LIN {X 0,Y 411.249,Z 344.255,A -85,B 0,C 180,E1 -10637.915,E2 -10637.915} C_VEL
LIN {X 0,Y 411.2,Z 344.267,A -85,B 0,C 180,E1 -10641.034,E2 -10641.034} C_VEL
LIN {X 0,Y 411.23,Z 344.259,A -85,B 0,C 180,E1 -10644.215,E2 -10644.215} C_VEL
LIN {X 0,Y 411.262,Z 344.258,A -85,B 0,C 180,E1 -10647.477,E2 -10647.477} C_VEL
LIN {X 0,Y 411.192,Z 344.266,A -85,B 0,C 180,E1 -10650.847,E2 -10650.847} C_VEL
LIN {X 0,Y 411.208,Z 344.262,A -85,B 0,C 180,E1 -10654.333,E2 -10654.333} C_VEL
LIN {X 0,Y 411.206,Z 344.261,A -85,B 0,C 180,E1 -10657.972,E2 -10657.972} C_VEL
LIN {X 0,Y 411.202,Z 344.264,A -85,B 0,C 180,E1 -10661.234,E2 -10661.234} C_VEL
LIN {X 0,Y 411.179,Z 344.268,A -85,B 0,C 180,E1 -10664.49,E2 -10664.49} C_VEL
LIN {X 0,Y 411.181,Z 344.267,A -85,B 0,C 180,E1 -10668.195,E2 -10668.195} C_VEL
LIN {X 0,Y 411.221,Z 344.265,A -85,B 0,C 180,E1 -10670.776,E2 -10670.776} C_VEL
LIN {X 0,Y 411.199,Z 344.267,A -85,B 0,C 180,E1 -10674.471,E2 -10674.471} C_VEL
LIN {X 0,Y 411.208,Z 344.263,A -85,B 0,C 180,E1 -10676.873,E2 -10676.873} C_VEL
LIN {X 0,Y 411.234,Z 344.26,A -85,B 0,C 180,E1 -10680.644,E2 -10680.644} C_VEL
LIN {X 0,Y 411.239,Z 344.259,A -85,B 0,C 180,E1 -10683.619,E2 -10683.619} C_VEL
LIN {X 0,Y 411.204,Z 344.264,A -85,B 0,C 180,E1 -10686.852,E2 -10686.852} C_VEL
LIN {X 0,Y 411.265,Z 344.256,A -85,B 0,C 180,E1 -10690.031,E2 -10690.031} C_VEL
LIN {X 0,Y 411.264,Z 344.254,A -85,B 0,C 180,E1 -10693.131,E2 -10693.131} C_VEL
LIN {X 0,Y 411.306,Z 344.251,A -85,B 0,C 180,E1 -10696.896,E2 -10696.896} C_VEL
LIN {X 0,Y 411.294,Z 344.253,A -85,B 0,C 180,E1 -10700.161,E2 -10700.161} C_VEL
LIN {X 0,Y 411.453,Z 344.232,A -85,B 0,C 180,E1 -10703.133,E2 -10703.133} C_VEL
LIN {X 0,Y 411.311,Z 344.249,A -85,B 0,C 180,E1 -10705.099,E2 -10705.099} C_VEL
LIN {X 0,Y 411.515,Z 344.228,A -85,B 0,C 180,E1 -10708.043,E2 -10708.043} C_VEL
LIN {X 0,Y 411.641,Z 344.212,A -85,B 0,C 180,E1 -10710,E2 -10710} C_VEL
LIN {X 0,Y 411.468,Z 344.229,A -85,B 0,C 180,E1 -10712.937,E2 -10712.937} C_VEL
LIN {X 0,Y 411.453,Z 344.232,A -85,B 0,C 180,E1 -10716.867,E2 -10716.867} C_VEL
LIN {X 0,Y 411.295,Z 344.253,A -85,B 0,C 180,E1 -10719.839,E2 -10719.839} C_VEL
LIN {X 0,Y 411.306,Z 344.25,A -85,B 0,C 180,E1 -10723.104,E2 -10723.104} C_VEL
LIN {X 0,Y 411.25,Z 344.255,A -85,B 0,C 180,E1 -10725.055,E2 -10725.055} C_VEL
LIN {X 0,Y 410.564,Z 344.346,A -85,B 0,C 180,E1 -10725.872,E2 -10725.872} C_VEL
LIN {X 0,Y 407.698,Z 344.703,A -85,B 0,C 180,E1 -10727.2,E2 -10727.2} C_VEL
LIN {X 0,Y 405.284,Z 345.005,A -85,B 0,C 180,E1 -10728.272,E2 -10728.272} C_VEL
LIN {X 0,Y 404.249,Z 345.131,A -85,B 0,C 180,E1 -10729.101,E2 -10729.101} C_VEL
LIN {X 0,Y 404.166,Z 345.14,A -85,B 0,C 180,E1 -10729.382,E2 -10729.382} C_VEL
LIN {X 0,Y 404.157,Z 345.141,A -85,B 0,C 180,E1 -10732.834,E2 -10732.834} C_VEL
LIN {X 0,Y 404.185,Z 345.139,A -85,B 0,C 180,E1 -10735.767,E2 -10735.767} C_VEL
LIN {X 0,Y 404.197,Z 345.137,A -85,B 0,C 180,E1 -10738,E2 -10738} C_VEL
LIN {X 0,Y 404.141,Z 345.146,A -85,B 0,C 180,E1 -10741.558,E2 -10741.558} C_VEL
LIN {X 0,Y 404.186,Z 345.137,A -85,B 0,C 180,E1 -10745.016,E2 -10745.016} C_VEL
LIN {X 0,Y 404.158,Z 345.141,A -85,B 0,C 180,E1 -10748.757,E2 -10748.757} C_VEL
LIN {X 0,Y 404.191,Z 345.138,A -85,B 0,C 180,E1 -10751.611,E2 -10751.611} C_VEL
LIN {X 0,Y 404.195,Z 345.136,A -85,B 0,C 180,E1 -10754.529,E2 -10754.529} C_VEL
LIN {X 0,Y 404.139,Z 345.146,A -85,B 0,C 180,E1 -10757.296,E2 -10757.296} C_VEL
LIN {X 0,Y 404.171,Z 345.137,A -85,B 0,C 180,E1 -10759.956,E2 -10759.956} C_VEL
LIN {X 0,Y 404.139,Z 345.146,A -85,B 0,C 180,E1 -10763.125,E2 -10763.125} C_VEL
LIN {X 0,Y 404.148,Z 345.141,A -85,B 0,C 180,E1 -10766.188,E2 -10766.188} C_VEL
LIN {X 0,Y 404.149,Z 345.142,A -85,B 0,C 180,E1 -10769.715,E2 -10769.715} C_VEL
LIN {X 0,Y 404.199,Z 345.138,A -85,B 0,C 180,E1 -10773.123,E2 -10773.123} C_VEL
LIN {X 0,Y 404.181,Z 345.139,A -85,B 0,C 180,E1 -10775.335,E2 -10775.335} C_VEL
LIN {X 0,Y 404.143,Z 345.143,A -85,B 0,C 180,E1 -10778.581,E2 -10778.581} C_VEL
LIN {X 0,Y 404.214,Z 345.132,A -85,B 0,C 180,E1 -10781.762,E2 -10781.762} C_VEL
LIN {X 0,Y 404.211,Z 345.135,A -85,B 0,C 180,E1 -10784.882,E2 -10784.882} C_VEL
LIN {X 0,Y 404.262,Z 345.128,A -85,B 0,C 180,E1 -10787.959,E2 -10787.959} C_VEL
LIN {X 0,Y 404.438,Z 345.106,A -85,B 0,C 180,E1 -10792.1,E2 -10792.1} C_VEL
LIN {X 0,Y 404.429,Z 345.107,A -85,B 0,C 180,E1 -10794.015,E2 -10794.015} C_VEL
LIN {X 0,Y 404.485,Z 345.099,A -85,B 0,C 180,E1 -10798.009,E2 -10798.009} C_VEL
LIN {X 0,Y 404.615,Z 345.084,A -85,B 0,C 180,E1 -10800,E2 -10800} C_VEL
LIN {X 0,Y 404.427,Z 345.108,A -85,B 0,C 180,E1 -10802.989,E2 -10802.989} C_VEL
LIN {X 0,Y 404.419,Z 345.11,A -85,B 0,C 180,E1 -10805.985,E2 -10805.985} C_VEL
LIN {X 0,Y 404.271,Z 345.127,A -85,B 0,C 180,E1 -10809.002,E2 -10809.002} C_VEL
LIN {X 0,Y 404.261,Z 345.129,A -85,B 0,C 180,E1 -10812.042,E2 -10812.042} C_VEL
LIN {X 0,Y 404.212,Z 345.132,A -85,B 0,C 180,E1 -10815.118,E2 -10815.118} C_VEL
LIN {X 0,Y 404.216,Z 345.136,A -85,B 0,C 180,E1 -10818.238,E2 -10818.238} C_VEL
LIN {X 0,Y 404.144,Z 345.143,A -85,B 0,C 180,E1 -10821.419,E2 -10821.419} C_VEL
LIN {X 0,Y 404.182,Z 345.139,A -85,B 0,C 180,E1 -10824.666,E2 -10824.666} C_VEL
LIN {X 0,Y 404.2,Z 345.137,A -85,B 0,C 180,E1 -10828,E2 -10828} C_VEL
LIN {X 0,Y 404.144,Z 345.142,A -85,B 0,C 180,E1 -10831.558,E2 -10831.558} C_VEL
LIN {X 0,Y 404.19,Z 345.135,A -85,B 0,C 180,E1 -10835.016,E2 -10835.016} C_VEL
LIN {X 0,Y 404.162,Z 345.14,A -85,B 0,C 180,E1 -10838.756,E2 -10838.756} C_VEL
LIN {X 0,Y 404.127,Z 345.146,A -85,B 0,C 180,E1 -10841.6,E2 -10841.6} C_VEL
LIN {X 0,Y 404.15,Z 345.145,A -85,B 0,C 180,E1 -10844.522,E2 -10844.522} C_VEL
LIN {X 0,Y 404.137,Z 345.204,A -85,B 0,C 180,E1 -10846.378,E2 -10846.378} C_VEL
LIN {X 0,Y 406.071,Z 354.648,A -85,B 0,C 180,E1 -10849.599,E2 -10849.599} C_VEL
LIN {X 0,Y 407.763,Z 363.407,A -85,B 0,C 180,E1 -10852.451,E2 -10852.451} C_VEL
LIN {X 0,Y 407.874,Z 366.908,A -85,B 0,C 180,E1 -10853.525,E2 -10853.525} C_VEL
LIN {X 0,Y 406.615,Z 380.772,A -85,B 0,C 180,E1 -10857.601,E2 -10857.601} C_VEL
LIN {X 0,Y 405.74,Z 392.561,A -85,B 0,C 180,E1 -10860.987,E2 -10860.987} C_VEL
LIN {X 0,Y 404.928,Z 405.007,A -85,B 0,C 180,E1 -10864.492,E2 -10864.492} C_VEL
LIN {X 0,Y 404.265,Z 417.836,A -85,B 0,C 180,E1 -10868.051,E2 -10868.051} C_VEL
LIN {X 0,Y 403.765,Z 431.296,A -85,B 0,C 180,E1 -10871.741,E2 -10871.741} C_VEL
LIN {X 0,Y 403.666,Z 434.163,A -85,B 0,C 180,E1 -10872.522,E2 -10872.522} C_VEL
LIN {X 0,Y 404.99,Z 448.876,A -85,B 0,C 180,E1 -10873.06,E2 -10873.06} C_VEL
LIN {X 0,Y 405.875,Z 461.695,A -85,B 0,C 180,E1 -10873.716,E2 -10873.716} C_VEL
LIN {X 0,Y 406.362,Z 472.774,A -85,B 0,C 180,E1 -10874.45,E2 -10874.45} C_VEL
LIN {X 0,Y 405.508,Z 484.977,A -85,B 0,C 180,E1 -10875.445,E2 -10875.445} C_VEL
LIN {X 0,Y 404.832,Z 495.687,A -85,B 0,C 180,E1 -10876.54,E2 -10876.54} C_VEL
LIN {X 0,Y 404.282,Z 504.941,A -85,B 0,C 180,E1 -10877.704,E2 -10877.704} C_VEL
LIN {X 0,Y 403.773,Z 514.717,A -85,B 0,C 180,E1 -10879.216,E2 -10879.216} C_VEL
LIN {X 0,Y 403.451,Z 522.561,A -85,B 0,C 180,E1 -10880.727,E2 -10880.727} C_VEL
LIN {X 0,Y 403.419,Z 527.916,A -85,B 0,C 180,E1 -10881.989,E2 -10881.989} C_VEL
LIN {X 0,Y 403.454,Z 533.164,A -85,B 0,C 180,E1 -10883.528,E2 -10883.528} C_VEL
LIN {X 0,Y 403.546,Z 537.03,A -85,B 0,C 180,E1 -10885.004,E2 -10885.004} C_VEL
LIN {X 0,Y 403.598,Z 539.018,A -85,B 0,C 180,E1 -10886.006,E2 -10886.006} C_VEL
LIN {X 0,Y 403.599,Z 540.55,A -85,B 0,C 180,E1 -10887.005,E2 -10887.005} C_VEL
LIN {X 0,Y 403.628,Z 541.647,A -85,B 0,C 180,E1 -10888.004,E2 -10888.004} C_VEL
LIN {X 0,Y 403.761,Z 542.278,A -85,B 0,C 180,E1 -10889.003,E2 -10889.003} C_VEL
LIN {X 0,Y 403.888,Z 542.48,A -85,B 0,C 180,E1 -10890,E2 -10890} C_VEL
LIN {X 0,Y 403.869,Z 542.237,A -85,B 0,C 180,E1 -10890.997,E2 -10890.997} C_VEL
LIN {X 0,Y 403.64,Z 541.526,A -85,B 0,C 180,E1 -10891.996,E2 -10891.996} C_VEL
LIN {X 0,Y 403.621,Z 540.374,A -85,B 0,C 180,E1 -10892.994,E2 -10892.994} C_VEL
LIN {X 0,Y 403.642,Z 537.838,A -85,B 0,C 180,E1 -10894.494,E2 -10894.494} C_VEL
LIN {X 0,Y 403.478,Z 534.22,A -85,B 0,C 180,E1 -10895.999,E2 -10895.999} C_VEL
LIN {X 0,Y 403.406,Z 529.478,A -85,B 0,C 180,E1 -10897.508,E2 -10897.508} C_VEL
LIN {X 0,Y 403.451,Z 523.498,A -85,B 0,C 180,E1 -10899.02,E2 -10899.02} C_VEL
LIN {X 0,Y 403.678,Z 516.15,A -85,B 0,C 180,E1 -10900.533,E2 -10900.533} C_VEL
LIN {X 0,Y 404.112,Z 507.171,A -85,B 0,C 180,E1 -10902.046,E2 -10902.046} C_VEL
LIN {X 0,Y 404.701,Z 497.278,A -85,B 0,C 180,E1 -10903.41,E2 -10903.41} C_VEL
LIN {X 0,Y 405.648,Z 486.03,A -85,B 0,C 180,E1 -10904.678,E2 -10904.678} C_VEL
LIN {X 0,Y 406.71,Z 473.812,A -85,B 0,C 180,E1 -10905.793,E2 -10905.793} C_VEL
LIN {X 0,Y 406.567,Z 460.164,A -85,B 0,C 180,E1 -10906.831,E2 -10906.831} C_VEL
LIN {X 0,Y 406.397,Z 447.657,A -85,B 0,C 180,E1 -10907.59,E2 -10907.59} C_VEL
LIN {X 0,Y 405.002,Z 433.311,A -85,B 0,C 180,E1 -10908.316,E2 -10908.316} C_VEL
LIN {X 0,Y 403.649,Z 424.626,A -85,B 0,C 180,E1 -10908.725,E2 -10908.725} C_VEL
LIN {X 0,Y 403.913,Z 413.212,A -85,B 0,C 180,E1 -10911.7,E2 -10911.7} C_VEL
LIN {X 0,Y 404.396,Z 399.615,A -85,B 0,C 180,E1 -10915.35,E2 -10915.35} C_VEL
LIN {X 0,Y 405,Z 386.397,A -85,B 0,C 180,E1 -10919.071,E2 -10919.071} C_VEL
LIN {X 0,Y 405.793,Z 375.051,A -85,B 0,C 180,E1 -10922.473,E2 -10922.473} C_VEL
LIN {X 0,Y 407.226,Z 362.64,A -85,B 0,C 180,E1 -10926.542,E2 -10926.542} C_VEL
LIN {X 0,Y 406.953,Z 359.119,A -85,B 0,C 180,E1 -10927.88,E2 -10927.88} C_VEL
LIN {X 0,Y 405.885,Z 353.328,A -85,B 0,C 180,E1 -10930.37,E2 -10930.37} C_VEL
LIN {X 0,Y 404.721,Z 347.779,A -85,B 0,C 180,E1 -10933.169,E2 -10933.169} C_VEL
LIN {X 0,Y 404.136,Z 345.147,A -85,B 0,C 180,E1 -10934.782,E2 -10934.782} C_VEL
LIN {X 0,Y 404.14,Z 345.146,A -85,B 0,C 180,E1 -10937.296,E2 -10937.296} C_VEL
LIN {X 0,Y 404.172,Z 345.142,A -85,B 0,C 180,E1 -10939.955,E2 -10939.955} C_VEL
LIN {X 0,Y 404.143,Z 345.145,A -85,B 0,C 180,E1 -10943.124,E2 -10943.124} C_VEL
LIN {X 0,Y 404.149,Z 345.144,A -85,B 0,C 180,E1 -10946.188,E2 -10946.188} C_VEL
LIN {X 0,Y 404.149,Z 345.144,A -85,B 0,C 180,E1 -10949.715,E2 -10949.715} C_VEL
LIN {X 0,Y 404.198,Z 345.136,A -85,B 0,C 180,E1 -10953.123,E2 -10953.123} C_VEL
LIN {X 0,Y 404.18,Z 345.139,A -85,B 0,C 180,E1 -10955.334,E2 -10955.334} C_VEL
LIN {X 0,Y 404.143,Z 345.145,A -85,B 0,C 180,E1 -10958.581,E2 -10958.581} C_VEL
LIN {X 0,Y 404.207,Z 345.241,A -85,B 0,C 180,E1 -10961.089,E2 -10961.089} C_VEL
LIN {X 0,Y 408.313,Z 356.062,A -85,B 0,C 180,E1 -10962.076,E2 -10962.076} C_VEL
LIN {X 0,Y 410.568,Z 363.518,A -85,B 0,C 180,E1 -10962.816,E2 -10962.816} C_VEL
LIN {X 0,Y 409.73,Z 376.006,A -85,B 0,C 180,E1 -10963.93,E2 -10963.93} C_VEL
LIN {X 0,Y 408.903,Z 386.087,A -85,B 0,C 180,E1 -10965.06,E2 -10965.06} C_VEL
LIN {X 0,Y 408.091,Z 395.094,A -85,B 0,C 180,E1 -10966.302,E2 -10966.302} C_VEL
LIN {X 0,Y 407.321,Z 402.523,A -85,B 0,C 180,E1 -10967.545,E2 -10967.545} C_VEL
LIN {X 0,Y 406.546,Z 409.803,A -85,B 0,C 180,E1 -10969.038,E2 -10969.038} C_VEL
LIN {X 0,Y 405.811,Z 416.513,A -85,B 0,C 180,E1 -10970.807,E2 -10970.807} C_VEL
LIN {X 0,Y 405.237,Z 421.446,A -85,B 0,C 180,E1 -10972.526,E2 -10972.526} C_VEL
LIN {X 0,Y 404.71,Z 424.575,A -85,B 0,C 180,E1 -10974.019,E2 -10974.019} C_VEL
LIN {X 0,Y 404.488,Z 426.074,A -85,B 0,C 180,E1 -10975.016,E2 -10975.016} C_VEL
LIN {X 0,Y 404.384,Z 427.144,A -85,B 0,C 180,E1 -10976.014,E2 -10976.014} C_VEL
LIN {X 0,Y 404.257,Z 427.831,A -85,B 0,C 180,E1 -10977.01,E2 -10977.01} C_VEL
LIN {X 0,Y 404.21,Z 428.103,A -85,B 0,C 180,E1 -10978.007,E2 -10978.007} C_VEL
LIN {X 0,Y 404.089,Z 427.417,A -85,B 0,C 180,E1 -10980,E2 -10980} C_VEL
LIN {X 0,Y 403.974,Z 426.508,A -85,B 0,C 180,E1 -10980.997,E2 -10980.997} C_VEL
LIN {X 0,Y 404.062,Z 425.133,A -85,B 0,C 180,E1 -10981.993,E2 -10981.993} C_VEL
LIN {X 0,Y 404.164,Z 422.298,A -85,B 0,C 180,E1 -10983.489,E2 -10983.489} C_VEL
LIN {X 0,Y 404.29,Z 418.443,A -85,B 0,C 180,E1 -10984.986,E2 -10984.986} C_VEL
LIN {X 0,Y 404.663,Z 413.44,A -85,B 0,C 180,E1 -10986.482,E2 -10986.482} C_VEL
LIN {X 0,Y 405.124,Z 407.168,A -85,B 0,C 180,E1 -10987.977,E2 -10987.977} C_VEL
LIN {X 0,Y 405.514,Z 399.438,A -85,B 0,C 180,E1 -10989.476,E2 -10989.476} C_VEL
LIN {X 0,Y 405.938,Z 391.594,A -85,B 0,C 180,E1 -10990.726,E2 -10990.726} C_VEL
LIN {X 0,Y 406.574,Z 382.084,A -85,B 0,C 180,E1 -10991.972,E2 -10991.972} C_VEL
LIN {X 0,Y 407.198,Z 370.353,A -85,B 0,C 180,E1 -10993.22,E2 -10993.22} C_VEL
LIN {X 0,Y 407.582,Z 360.495,A -85,B 0,C 180,E1 -10994.072,E2 -10994.072} C_VEL
LIN {X 0,Y 407.621,Z 358.036,A -85,B 0,C 180,E1 -10994.26,E2 -10994.26} C_VEL
LIN {X 0,Y 404.235,Z 345.134,A -85,B 0,C 180,E1 -10995.246,E2 -10995.246} C_VEL
LIN {X 0,Y 404.208,Z 345.132,A -85,B 0,C 180,E1 -10998.238,E2 -10998.238} C_VEL
LIN {X 0,Y 404.142,Z 345.143,A -85,B 0,C 180,E1 -11001.419,E2 -11001.419} C_VEL
LIN {X 0,Y 404.18,Z 345.14,A -85,B 0,C 180,E1 -11004.665,E2 -11004.665} C_VEL
LIN {X 0,Y 404.198,Z 345.135,A -85,B 0,C 180,E1 -11007.999,E2 -11007.999} C_VEL
LIN {X 0,Y 404.142,Z 345.143,A -85,B 0,C 180,E1 -11011.558,E2 -11011.558} C_VEL
LIN {X 0,Y 404.187,Z 345.14,A -85,B 0,C 180,E1 -11015.016,E2 -11015.016} C_VEL
LIN {X 0,Y 404.166,Z 345.143,A -85,B 0,C 180,E1 -11018.756,E2 -11018.756} C_VEL
LIN {X 0,Y 404.152,Z 345.141,A -85,B 0,C 180,E1 -11021.604,E2 -11021.604} C_VEL
LIN {X 0,Y 404.148,Z 345.144,A -85,B 0,C 180,E1 -11024.522,E2 -11024.522} C_VEL
LIN {X 0,Y 404.142,Z 345.143,A -85,B 0,C 180,E1 -11027.296,E2 -11027.296} C_VEL
LIN {X 0,Y 404.17,Z 345.139,A -85,B 0,C 180,E1 -11029.955,E2 -11029.955} C_VEL
LIN {X 0,Y 404.138,Z 345.142,A -85,B 0,C 180,E1 -11033.125,E2 -11033.125} C_VEL
LIN {X 0,Y 404.146,Z 345.143,A -85,B 0,C 180,E1 -11036.188,E2 -11036.188} C_VEL
LIN {X 0,Y 404.147,Z 345.142,A -85,B 0,C 180,E1 -11039.715,E2 -11039.715} C_VEL
LIN {X 0,Y 404.196,Z 345.136,A -85,B 0,C 180,E1 -11043.123,E2 -11043.123} C_VEL
LIN {X 0,Y 404.178,Z 345.138,A -85,B 0,C 180,E1 -11045.334,E2 -11045.334} C_VEL
LIN {X 0,Y 404.164,Z 345.143,A -85,B 0,C 180,E1 -11048.582,E2 -11048.582} C_VEL
LIN {X 0,Y 404.215,Z 345.132,A -85,B 0,C 180,E1 -11051.762,E2 -11051.762} C_VEL
LIN {X 0,Y 404.207,Z 345.134,A -85,B 0,C 180,E1 -11054.882,E2 -11054.882} C_VEL
LIN {X 0,Y 404.258,Z 345.131,A -85,B 0,C 180,E1 -11057.959,E2 -11057.959} C_VEL
LIN {X 0,Y 404.405,Z 345.111,A -85,B 0,C 180,E1 -11062.129,E2 -11062.129} C_VEL
LIN {X 0,Y 404.421,Z 345.109,A -85,B 0,C 180,E1 -11064.015,E2 -11064.015} C_VEL
LIN {X 0,Y 404.484,Z 345.103,A -85,B 0,C 180,E1 -11068.009,E2 -11068.009} C_VEL
LIN {X 0,Y 404.611,Z 345.088,A -85,B 0,C 180,E1 -11070,E2 -11070} C_VEL
LIN {X 0,Y 404.425,Z 345.106,A -85,B 0,C 180,E1 -11072.988,E2 -11072.988} C_VEL
LIN {X 0,Y 404.4,Z 345.11,A -85,B 0,C 180,E1 -11076.988,E2 -11076.988} C_VEL
LIN {X 0,Y 404.26,Z 345.13,A -85,B 0,C 180,E1 -11080.012,E2 -11080.012} C_VEL
LIN {X 0,Y 404.267,Z 345.127,A -85,B 0,C 180,E1 -11083.212,E2 -11083.212} C_VEL
LIN {X 0,Y 404.217,Z 345.131,A -85,B 0,C 180,E1 -11087.007,E2 -11087.007} C_VEL
LIN {X 0,Y 404.166,Z 345.14,A -85,B 0,C 180,E1 -11089.382,E2 -11089.382} C_VEL
LIN {X 0,Y 403.495,Z 345.223,A -85,B 0,C 180,E1 -11090.213,E2 -11090.213} C_VEL
LIN {X 0,Y 400.631,Z 345.583,A -85,B 0,C 180,E1 -11091.564,E2 -11091.564} C_VEL
LIN {X 0,Y 398.217,Z 345.881,A -85,B 0,C 180,E1 -11092.655,E2 -11092.655} C_VEL
LIN {X 0,Y 397.198,Z 346.01,A -85,B 0,C 180,E1 -11093.499,E2 -11093.499} C_VEL
LIN {X 0,Y 397.124,Z 346.017,A -85,B 0,C 180,E1 -11093.785,E2 -11093.785} C_VEL
LIN {X 0,Y 397.196,Z 346.009,A -85,B 0,C 180,E1 -11097.39,E2 -11097.39} C_VEL
LIN {X 0,Y 397.08,Z 346.022,A -85,B 0,C 180,E1 -11100.883,E2 -11100.883} C_VEL
LIN {X 0,Y 397.127,Z 346.014,A -85,B 0,C 180,E1 -11104.494,E2 -11104.494} C_VEL
LIN {X 0,Y 397.105,Z 346.018,A -85,B 0,C 180,E1 -11108.275,E2 -11108.275} C_VEL
LIN {X 0,Y 397.157,Z 346.013,A -85,B 0,C 180,E1 -11111.993,E2 -11111.993} C_VEL
LIN {X 0,Y 397.114,Z 346.02,A -85,B 0,C 180,E1 -11115.065,E2 -11115.065} C_VEL
LIN {X 0,Y 397.068,Z 346.023,A -85,B 0,C 180,E1 -11118.021,E2 -11118.021} C_VEL
LIN {X 0,Y 397.132,Z 346.019,A -85,B 0,C 180,E1 -11121.139,E2 -11121.139} C_VEL
LIN {X 0,Y 397.122,Z 346.017,A -85,B 0,C 180,E1 -11124.497,E2 -11124.497} C_VEL
LIN {X 0,Y 397.081,Z 346.022,A -85,B 0,C 180,E1 -11127.929,E2 -11127.929} C_VEL
LIN {X 0,Y 397.126,Z 346.018,A -85,B 0,C 180,E1 -11131.457,E2 -11131.457} C_VEL
LIN {X 0,Y 397.157,Z 346.014,A -85,B 0,C 180,E1 -11134.488,E2 -11134.488} C_VEL
LIN {X 0,Y 397.113,Z 346.021,A -85,B 0,C 180,E1 -11137.086,E2 -11137.086} C_VEL
LIN {X 0,Y 397.152,Z 346.013,A -85,B 0,C 180,E1 -11140.353,E2 -11140.353} C_VEL
LIN {X 0,Y 397.171,Z 346.01,A -85,B 0,C 180,E1 -11143.553,E2 -11143.553} C_VEL
LIN {X 0,Y 397.233,Z 346.005,A -85,B 0,C 180,E1 -11146.703,E2 -11146.703} C_VEL
LIN {X 0,Y 397.223,Z 346.004,A -85,B 0,C 180,E1 -11149.809,E2 -11149.809} C_VEL
LIN {X 0,Y 397.369,Z 345.989,A -85,B 0,C 180,E1 -11152.888,E2 -11152.888} C_VEL
LIN {X 0,Y 397.258,Z 346.001,A -85,B 0,C 180,E1 -11154.925,E2 -11154.925} C_VEL
LIN {X 0,Y 397.454,Z 345.975,A -85,B 0,C 180,E1 -11157.973,E2 -11157.973} C_VEL
LIN {X 0,Y 397.584,Z 345.96,A -85,B 0,C 180,E1 -11160,E2 -11160} C_VEL
LIN {X 0,Y 397.386,Z 345.985,A -85,B 0,C 180,E1 -11163.042,E2 -11163.042} C_VEL
LIN {X 0,Y 397.369,Z 345.988,A -85,B 0,C 180,E1 -11166.092,E2 -11166.092} C_VEL
LIN {X 0,Y 397.241,Z 346.002,A -85,B 0,C 180,E1 -11169.162,E2 -11169.162} C_VEL
LIN {X 0,Y 397.224,Z 346.007,A -85,B 0,C 180,E1 -11172.258,E2 -11172.258} C_VEL
LIN {X 0,Y 397.184,Z 346.007,A -85,B 0,C 180,E1 -11175.392,E2 -11175.392} C_VEL
LIN {X 0,Y 397.168,Z 346.012,A -85,B 0,C 180,E1 -11178.573,E2 -11178.573} C_VEL
LIN {X 0,Y 397.102,Z 346.022,A -85,B 0,C 180,E1 -11181.818,E2 -11181.818} C_VEL
LIN {X 0,Y 397.161,Z 346.012,A -85,B 0,C 180,E1 -11185.132,E2 -11185.132} C_VEL
LIN {X 0,Y 397.166,Z 346.013,A -85,B 0,C 180,E1 -11187.776,E2 -11187.776} C_VEL
LIN {X 0,Y 397.083,Z 346.02,A -85,B 0,C 180,E1 -11190.882,E2 -11190.882} C_VEL
LIN {X 0,Y 397.13,Z 346.016,A -85,B 0,C 180,E1 -11194.493,E2 -11194.493} C_VEL
LIN {X 0,Y 397.11,Z 346.02,A -85,B 0,C 180,E1 -11198.274,E2 -11198.274} C_VEL
LIN {X 0,Y 397.093,Z 346.02,A -85,B 0,C 180,E1 -11200.909,E2 -11200.909} C_VEL
LIN {X 0,Y 397.105,Z 346.021,A -85,B 0,C 180,E1 -11203.648,E2 -11203.648} C_VEL
LIN {X 0,Y 397.121,Z 346.135,A -85,B 0,C 180,E1 -11206.109,E2 -11206.109} C_VEL
LIN {X 0,Y 399.149,Z 356.213,A -85,B 0,C 180,E1 -11209.598,E2 -11209.598} C_VEL
LIN {X 0,Y 400.825,Z 364.863,A -85,B 0,C 180,E1 -11212.465,E2 -11212.465} C_VEL
LIN {X 0,Y 400.894,Z 367.885,A -85,B 0,C 180,E1 -11213.412,E2 -11213.412} C_VEL
LIN {X 0,Y 399.657,Z 380.975,A -85,B 0,C 180,E1 -11217.333,E2 -11217.333} C_VEL
LIN {X 0,Y 398.657,Z 393.5,A -85,B 0,C 180,E1 -11221,E2 -11221} C_VEL
LIN {X 0,Y 397.789,Z 407.111,A -85,B 0,C 180,E1 -11224.911,E2 -11224.911} C_VEL
LIN {X 0,Y 397.141,Z 418.69,A -85,B 0,C 180,E1 -11228.184,E2 -11228.184} C_VEL
LIN {X 0,Y 396.705,Z 430.173,A -85,B 0,C 180,E1 -11231.404,E2 -11231.404} C_VEL
LIN {X 0,Y 396.615,Z 433.284,A -85,B 0,C 180,E1 -11232.268,E2 -11232.268} C_VEL
LIN {X 0,Y 397.959,Z 449.198,A -85,B 0,C 180,E1 -11232.885,E2 -11232.885} C_VEL
LIN {X 0,Y 398.9,Z 462.726,A -85,B 0,C 180,E1 -11233.626,E2 -11233.626} C_VEL
LIN {X 0,Y 399.353,Z 472.476,A -85,B 0,C 180,E1 -11234.301,E2 -11234.301} C_VEL
LIN {X 0,Y 398.478,Z 484.535,A -85,B 0,C 180,E1 -11235.313,E2 -11235.313} C_VEL
LIN {X 0,Y 397.77,Z 495.235,A -85,B 0,C 180,E1 -11236.441,E2 -11236.441} C_VEL
LIN {X 0,Y 397.321,Z 503.419,A -85,B 0,C 180,E1 -11237.485,E2 -11237.485} C_VEL
LIN {X 0,Y 396.846,Z 511.786,A -85,B 0,C 180,E1 -11238.766,E2 -11238.766} C_VEL
LIN {X 0,Y 396.483,Z 519.997,A -85,B 0,C 180,E1 -11240.305,E2 -11240.305} C_VEL
LIN {X 0,Y 396.365,Z 526.615,A -85,B 0,C 180,E1 -11241.845,E2 -11241.845} C_VEL
LIN {X 0,Y 396.346,Z 531.319,A -85,B 0,C 180,E1 -11243.214,E2 -11243.214} C_VEL
LIN {X 0,Y 396.502,Z 535.858,A -85,B 0,C 180,E1 -11244.915,E2 -11244.915} C_VEL
LIN {X 0,Y 396.562,Z 537.875,A -85,B 0,C 180,E1 -11245.935,E2 -11245.935} C_VEL
LIN {X 0,Y 396.568,Z 539.427,A -85,B 0,C 180,E1 -11246.952,E2 -11246.952} C_VEL
LIN {X 0,Y 396.601,Z 540.548,A -85,B 0,C 180,E1 -11247.969,E2 -11247.969} C_VEL
LIN {X 0,Y 396.746,Z 541.214,A -85,B 0,C 180,E1 -11248.985,E2 -11248.985} C_VEL
LIN {X 0,Y 396.888,Z 541.43,A -85,B 0,C 180,E1 -11250,E2 -11250} C_VEL
LIN {X 0,Y 396.841,Z 541.195,A -85,B 0,C 180,E1 -11251.015,E2 -11251.015} C_VEL
LIN {X 0,Y 396.602,Z 540.504,A -85,B 0,C 180,E1 -11252.031,E2 -11252.031} C_VEL
LIN {X 0,Y 396.579,Z 539.371,A -85,B 0,C 180,E1 -11253.048,E2 -11253.048} C_VEL
LIN {X 0,Y 396.568,Z 536.858,A -85,B 0,C 180,E1 -11254.574,E2 -11254.574} C_VEL
LIN {X 0,Y 396.42,Z 533.266,A -85,B 0,C 180,E1 -11256.106,E2 -11256.106} C_VEL
LIN {X 0,Y 396.334,Z 528.555,A -85,B 0,C 180,E1 -11257.643,E2 -11257.643} C_VEL
LIN {X 0,Y 396.414,Z 521.495,A -85,B 0,C 180,E1 -11259.439,E2 -11259.439} C_VEL
LIN {X 0,Y 396.722,Z 513.972,A -85,B 0,C 180,E1 -11260.978,E2 -11260.978} C_VEL
LIN {X 0,Y 397.273,Z 504.757,A -85,B 0,C 180,E1 -11262.516,E2 -11262.516} C_VEL
LIN {X 0,Y 397.828,Z 495.743,A -85,B 0,C 180,E1 -11263.765,E2 -11263.765} C_VEL
LIN {X 0,Y 398.84,Z 484.382,A -85,B 0,C 180,E1 -11265.065,E2 -11265.065} C_VEL
LIN {X 0,Y 399.877,Z 472.122,A -85,B 0,C 180,E1 -11266.201,E2 -11266.201} C_VEL
LIN {X 0,Y 399.771,Z 460.39,A -85,B 0,C 180,E1 -11267.126,E2 -11267.126} C_VEL
LIN {X 0,Y 399.67,Z 448.123,A -85,B 0,C 180,E1 -11267.915,E2 -11267.915} C_VEL
LIN {X 0,Y 398.355,Z 434.155,A -85,B 0,C 180,E1 -11268.683,E2 -11268.683} C_VEL
LIN {X 0,Y 396.608,Z 423.201,A -85,B 0,C 180,E1 -11269.204,E2 -11269.204} C_VEL
LIN {X 0,Y 396.889,Z 411.342,A -85,B 0,C 180,E1 -11272.378,E2 -11272.378} C_VEL
LIN {X 0,Y 397.409,Z 398.777,A -85,B 0,C 180,E1 -11275.853,E2 -11275.853} C_VEL
LIN {X 0,Y 398.088,Z 385.79,A -85,B 0,C 180,E1 -11279.625,E2 -11279.625} C_VEL
LIN {X 0,Y 398.985,Z 374.62,A -85,B 0,C 180,E1 -11283.097,E2 -11283.097} C_VEL
LIN {X 0,Y 400.335,Z 364.139,A -85,B 0,C 180,E1 -11286.647,E2 -11286.647} C_VEL
LIN {X 0,Y 400.079,Z 360.824,A -85,B 0,C 180,E1 -11287.94,E2 -11287.94} C_VEL
LIN {X 0,Y 399.242,Z 356.124,A -85,B 0,C 180,E1 -11289.98,E2 -11289.98} C_VEL
LIN {X 0,Y 398.058,Z 350.351,A -85,B 0,C 180,E1 -11292.886,E2 -11292.886} C_VEL
LIN {X 0,Y 397.104,Z 346.021,A -85,B 0,C 180,E1 -11295.53,E2 -11295.53} C_VEL
LIN {X 0,Y 397.092,Z 346.021,A -85,B 0,C 180,E1 -11299.091,E2 -11299.091} C_VEL
LIN {X 0,Y 397.108,Z 346.02,A -85,B 0,C 180,E1 -11301.725,E2 -11301.725} C_VEL
LIN {X 0,Y 397.13,Z 346.016,A -85,B 0,C 180,E1 -11305.507,E2 -11305.507} C_VEL
LIN {X 0,Y 397.082,Z 346.023,A -85,B 0,C 180,E1 -11309.118,E2 -11309.118} C_VEL
LIN {X 0,Y 397.198,Z 346.009,A -85,B 0,C 180,E1 -11312.61,E2 -11312.61} C_VEL
LIN {X 0,Y 397.136,Z 346.018,A -85,B 0,C 180,E1 -11315.982,E2 -11315.982} C_VEL
LIN {X 0,Y 397.143,Z 346.018,A -85,B 0,C 180,E1 -11319.705,E2 -11319.705} C_VEL
LIN {X 0,Y 397.157,Z 346.071,A -85,B 0,C 180,E1 -11320.555,E2 -11320.555} C_VEL
LIN {X 0,Y 398.185,Z 348.893,A -85,B 0,C 180,E1 -11320.808,E2 -11320.808} C_VEL
LIN {X 0,Y 401.977,Z 358.567,A -85,B 0,C 180,E1 -11321.773,E2 -11321.773} C_VEL
LIN {X 0,Y 404.093,Z 365.705,A -85,B 0,C 180,E1 -11322.511,E2 -11322.511} C_VEL
LIN {X 0,Y 403.269,Z 376.91,A -85,B 0,C 180,E1 -11323.538,E2 -11323.538} C_VEL
LIN {X 0,Y 402.399,Z 386.348,A -85,B 0,C 180,E1 -11324.602,E2 -11324.602} C_VEL
LIN {X 0,Y 401.41,Z 396.781,A -85,B 0,C 180,E1 -11326.07,E2 -11326.07} C_VEL
LIN {X 0,Y 400.574,Z 404.135,A -85,B 0,C 180,E1 -11327.331,E2 -11327.331} C_VEL
LIN {X 0,Y 399.749,Z 411.327,A -85,B 0,C 180,E1 -11328.849,E2 -11328.849} C_VEL
LIN {X 0,Y 398.992,Z 417.588,A -85,B 0,C 180,E1 -11330.544,E2 -11330.544} C_VEL
LIN {X 0,Y 398.318,Z 422.751,A -85,B 0,C 180,E1 -11332.395,E2 -11332.395} C_VEL
LIN {X 0,Y 397.759,Z 425.821,A -85,B 0,C 180,E1 -11333.914,E2 -11333.914} C_VEL
LIN {X 0,Y 397.531,Z 427.281,A -85,B 0,C 180,E1 -11334.929,E2 -11334.929} C_VEL
LIN {X 0,Y 397.401,Z 428.323,A -85,B 0,C 180,E1 -11335.943,E2 -11335.943} C_VEL
LIN {X 0,Y 397.278,Z 428.977,A -85,B 0,C 180,E1 -11336.958,E2 -11336.958} C_VEL
LIN {X 0,Y 397.206,Z 429.203,A -85,B 0,C 180,E1 -11337.972,E2 -11337.972} C_VEL
LIN {X 0,Y 397.124,Z 429.023,A -85,B 0,C 180,E1 -11338.986,E2 -11338.986} C_VEL
LIN {X 0,Y 397.073,Z 428.452,A -85,B 0,C 180,E1 -11340,E2 -11340} C_VEL
LIN {X 0,Y 396.95,Z 427.499,A -85,B 0,C 180,E1 -11341.014,E2 -11341.014} C_VEL
LIN {X 0,Y 397.038,Z 426.073,A -85,B 0,C 180,E1 -11342.029,E2 -11342.029} C_VEL
LIN {X 0,Y 397.145,Z 423.173,A -85,B 0,C 180,E1 -11343.551,E2 -11343.551} C_VEL
LIN {X 0,Y 397.28,Z 419.253,A -85,B 0,C 180,E1 -11345.074,E2 -11345.074} C_VEL
LIN {X 0,Y 397.674,Z 414.183,A -85,B 0,C 180,E1 -11346.596,E2 -11346.596} C_VEL
LIN {X 0,Y 398.133,Z 407.849,A -85,B 0,C 180,E1 -11348.118,E2 -11348.118} C_VEL
LIN {X 0,Y 398.534,Z 400.044,A -85,B 0,C 180,E1 -11349.644,E2 -11349.644} C_VEL
LIN {X 0,Y 399.001,Z 392.102,A -85,B 0,C 180,E1 -11350.915,E2 -11350.915} C_VEL
LIN {X 0,Y 399.639,Z 382.463,A -85,B 0,C 180,E1 -11352.183,E2 -11352.183} C_VEL
LIN {X 0,Y 400.3,Z 370.61,A -85,B 0,C 180,E1 -11353.452,E2 -11353.452} C_VEL
LIN {X 0,Y 400.633,Z 359.238,A -85,B 0,C 180,E1 -11354.426,E2 -11354.426} C_VEL
LIN {X 0,Y 397.436,Z 347.091,A -85,B 0,C 180,E1 -11355.382,E2 -11355.382} C_VEL
LIN {X 0,Y 397.202,Z 346.009,A -85,B 0,C 180,E1 -11355.49,E2 -11355.49} C_VEL
LIN {X 0,Y 397.161,Z 346.011,A -85,B 0,C 180,E1 -11358.573,E2 -11358.573} C_VEL
LIN {X 0,Y 397.1,Z 346.019,A -85,B 0,C 180,E1 -11361.818,E2 -11361.818} C_VEL
LIN {X 0,Y 397.16,Z 346.014,A -85,B 0,C 180,E1 -11365.131,E2 -11365.131} C_VEL
LIN {X 0,Y 397.165,Z 346.012,A -85,B 0,C 180,E1 -11367.776,E2 -11367.776} C_VEL
LIN {X 0,Y 397.081,Z 346.024,A -85,B 0,C 180,E1 -11370.882,E2 -11370.882} C_VEL
LIN {X 0,Y 397.128,Z 346.016,A -85,B 0,C 180,E1 -11374.493,E2 -11374.493} C_VEL
LIN {X 0,Y 397.112,Z 346.018,A -85,B 0,C 180,E1 -11378.274,E2 -11378.274} C_VEL
LIN {X 0,Y 397.115,Z 346.02,A -85,B 0,C 180,E1 -11380.905,E2 -11380.905} C_VEL
LIN {X 0,Y 397.104,Z 346.019,A -85,B 0,C 180,E1 -11383.648,E2 -11383.648} C_VEL
LIN {X 0,Y 397.107,Z 346.02,A -85,B 0,C 180,E1 -11386.52,E2 -11386.52} C_VEL
LIN {X 0,Y 397.115,Z 346.019,A -85,B 0,C 180,E1 -11390.423,E2 -11390.423} C_VEL
LIN {X 0,Y 397.109,Z 346.019,A -85,B 0,C 180,E1 -11394.265,E2 -11394.265} C_VEL
LIN {X 0,Y 397.115,Z 346.019,A -85,B 0,C 180,E1 -11396.727,E2 -11396.727} C_VEL
LIN {X 0,Y 397.125,Z 346.019,A -85,B 0,C 180,E1 -11400.296,E2 -11400.296} C_VEL
LIN {X 0,Y 397.195,Z 346.01,A -85,B 0,C 180,E1 -11402.61,E2 -11402.61} C_VEL
LIN {X 0,Y 397.134,Z 346.017,A -85,B 0,C 180,E1 -11405.982,E2 -11405.982} C_VEL
LIN {X 0,Y 397.155,Z 346.012,A -85,B 0,C 180,E1 -11409.698,E2 -11409.698} C_VEL
LIN {X 0,Y 397.183,Z 346.009,A -85,B 0,C 180,E1 -11412.845,E2 -11412.845} C_VEL
LIN {X 0,Y 397.229,Z 346.005,A -85,B 0,C 180,E1 -11416.703,E2 -11416.703} C_VEL
LIN {X 0,Y 397.219,Z 346.008,A -85,B 0,C 180,E1 -11419.809,E2 -11419.809} C_VEL
LIN {X 0,Y 397.35,Z 345.988,A -85,B 0,C 180,E1 -11422.888,E2 -11422.888} C_VEL
LIN {X 0,Y 397.255,Z 346,A -85,B 0,C 180,E1 -11424.925,E2 -11424.925} C_VEL
LIN {X 0,Y 397.453,Z 345.979,A -85,B 0,C 180,E1 -11427.973,E2 -11427.973} C_VEL
LIN {X 0,Y 397.58,Z 345.964,A -85,B 0,C 180,E1 -11430,E2 -11430} C_VEL
LIN {X 0,Y 397.383,Z 345.984,A -85,B 0,C 180,E1 -11433.041,E2 -11433.041} C_VEL
LIN {X 0,Y 397.372,Z 345.987,A -85,B 0,C 180,E1 -11436.092,E2 -11436.092} C_VEL
LIN {X 0,Y 397.254,Z 346.001,A -85,B 0,C 180,E1 -11439.162,E2 -11439.162} C_VEL
LIN {X 0,Y 397.221,Z 346.006,A -85,B 0,C 180,E1 -11442.258,E2 -11442.258} C_VEL
LIN {X 0,Y 397.181,Z 346.01,A -85,B 0,C 180,E1 -11445.392,E2 -11445.392} C_VEL
LIN {X 0,Y 397.164,Z 346.01,A -85,B 0,C 180,E1 -11448.574,E2 -11448.574} C_VEL
LIN {X 0,Y 397.11,Z 346.02,A -85,B 0,C 180,E1 -11451.818,E2 -11451.818} C_VEL
LIN {X 0,Y 397.124,Z 346.017,A -85,B 0,C 180,E1 -11453.785,E2 -11453.785} C_VEL
LIN {X 0,Y 396.488,Z 346.1,A -85,B 0,C 180,E1 -11454.632,E2 -11454.632} C_VEL
LIN {X 0,Y 393.665,Z 346.454,A -85,B 0,C 180,E1 -11456.009,E2 -11456.009} C_VEL
LIN {X 0,Y 391.242,Z 346.754,A -85,B 0,C 180,E1 -11457.121,E2 -11457.121} C_VEL
LIN {X 0,Y 390.176,Z 346.884,A -85,B 0,C 180,E1 -11457.981,E2 -11457.981} C_VEL
LIN {X 0,Y 390.076,Z 346.894,A -85,B 0,C 180,E1 -11458.273,E2 -11458.273} C_VEL
LIN {X 0,Y 390.025,Z 346.904,A -85,B 0,C 180,E1 -11461.505,E2 -11461.505} C_VEL
LIN {X 0,Y 390.086,Z 346.895,A -85,B 0,C 180,E1 -11465.207,E2 -11465.207} C_VEL
LIN {X 0,Y 390.072,Z 346.898,A -85,B 0,C 180,E1 -11469.219,E2 -11469.219} C_VEL
LIN {X 0,Y 390.123,Z 346.888,A -85,B 0,C 180,E1 -11472.387,E2 -11472.387} C_VEL
LIN {X 0,Y 390.064,Z 346.899,A -85,B 0,C 180,E1 -11475.357,E2 -11475.357} C_VEL
LIN {X 0,Y 390.033,Z 346.899,A -85,B 0,C 180,E1 -11478.187,E2 -11478.187} C_VEL
LIN {X 0,Y 390.092,Z 346.894,A -85,B 0,C 180,E1 -11480.908,E2 -11480.908} C_VEL
LIN {X 0,Y 390.088,Z 346.895,A -85,B 0,C 180,E1 -11484.794,E2 -11484.794} C_VEL
LIN {X 0,Y 390.027,Z 346.902,A -85,B 0,C 180,E1 -11488.496,E2 -11488.496} C_VEL
LIN {X 0,Y 390.12,Z 346.889,A -85,B 0,C 180,E1 -11492.07,E2 -11492.07} C_VEL
LIN {X 0,Y 390.084,Z 346.893,A -85,B 0,C 180,E1 -11495.52,E2 -11495.52} C_VEL
LIN {X 0,Y 390.06,Z 346.901,A -85,B 0,C 180,E1 -11498.878,E2 -11498.878} C_VEL
LIN {X 0,Y 390.132,Z 346.887,A -85,B 0,C 180,E1 -11502.167,E2 -11502.167} C_VEL
LIN {X 0,Y 390.149,Z 346.886,A -85,B 0,C 180,E1 -11505.393,E2 -11505.393} C_VEL
LIN {X 0,Y 390.154,Z 346.887,A -85,B 0,C 180,E1 -11508.571,E2 -11508.571} C_VEL
LIN {X 0,Y 390.349,Z 346.861,A -85,B 0,C 180,E1 -11511.993,E2 -11511.993} C_VEL
LIN {X 0,Y 390.23,Z 346.878,A -85,B 0,C 180,E1 -11514.834,E2 -11514.834} C_VEL
LIN {X 0,Y 390.423,Z 346.85,A -85,B 0,C 180,E1 -11517.937,E2 -11517.937} C_VEL
LIN {X 0,Y 390.554,Z 346.835,A -85,B 0,C 180,E1 -11520,E2 -11520} C_VEL
LIN {X 0,Y 390.32,Z 346.865,A -85,B 0,C 180,E1 -11523.097,E2 -11523.097} C_VEL
LIN {X 0,Y 390.322,Z 346.866,A -85,B 0,C 180,E1 -11526.202,E2 -11526.202} C_VEL
LIN {X 0,Y 390.198,Z 346.879,A -85,B 0,C 180,E1 -11529.329,E2 -11529.329} C_VEL
LIN {X 0,Y 390.176,Z 346.885,A -85,B 0,C 180,E1 -11532.483,E2 -11532.483} C_VEL
LIN {X 0,Y 390.144,Z 346.885,A -85,B 0,C 180,E1 -11535.677,E2 -11535.677} C_VEL
LIN {X 0,Y 390.111,Z 346.89,A -85,B 0,C 180,E1 -11538.922,E2 -11538.922} C_VEL
LIN {X 0,Y 390.045,Z 346.9,A -85,B 0,C 180,E1 -11542.234,E2 -11542.234} C_VEL
LIN {X 0,Y 390.124,Z 346.89,A -85,B 0,C 180,E1 -11545.743,E2 -11545.743} C_VEL
LIN {X 0,Y 390.063,Z 346.895,A -85,B 0,C 180,E1 -11549.109,E2 -11549.109} C_VEL
LIN {X 0,Y 390.047,Z 346.896,A -85,B 0,C 180,E1 -11552.721,E2 -11552.721} C_VEL
LIN {X 0,Y 390.062,Z 346.9,A -85,B 0,C 180,E1 -11555.826,E2 -11555.826} C_VEL
LIN {X 0,Y 390.075,Z 346.895,A -85,B 0,C 180,E1 -11559.219,E2 -11559.219} C_VEL
LIN {X 0,Y 390.046,Z 346.901,A -85,B 0,C 180,E1 -11562.374,E2 -11562.374} C_VEL
LIN {X 0,Y 390.08,Z 346.946,A -85,B 0,C 180,E1 -11565.792,E2 -11565.792} C_VEL
LIN {X 0,Y 392.073,Z 357.05,A -85,B 0,C 180,E1 -11569.366,E2 -11569.366} C_VEL
LIN {X 0,Y 393.734,Z 365.542,A -85,B 0,C 180,E1 -11572.233,E2 -11572.233} C_VEL
LIN {X 0,Y 393.885,Z 369.214,A -85,B 0,C 180,E1 -11573.411,E2 -11573.411} C_VEL
LIN {X 0,Y 392.543,Z 382.655,A -85,B 0,C 180,E1 -11577.512,E2 -11577.512} C_VEL
LIN {X 0,Y 391.584,Z 394.401,A -85,B 0,C 180,E1 -11581.014,E2 -11581.014} C_VEL
LIN {X 0,Y 390.676,Z 407.962,A -85,B 0,C 180,E1 -11584.991,E2 -11584.991} C_VEL
LIN {X 0,Y 390.02,Z 419.5,A -85,B 0,C 180,E1 -11588.321,E2 -11588.321} C_VEL
LIN {X 0,Y 389.551,Z 432.357,A -85,B 0,C 180,E1 -11592.003,E2 -11592.003} C_VEL
LIN {X 0,Y 389.702,Z 434.614,A -85,B 0,C 180,E1 -11592.112,E2 -11592.112} C_VEL
LIN {X 0,Y 390.864,Z 448.589,A -85,B 0,C 180,E1 -11592.67,E2 -11592.67} C_VEL
LIN {X 0,Y 391.759,Z 461.392,A -85,B 0,C 180,E1 -11593.386,E2 -11593.386} C_VEL
LIN {X 0,Y 392.304,Z 472.096,A -85,B 0,C 180,E1 -11594.145,E2 -11594.145} C_VEL
LIN {X 0,Y 391.45,Z 484.035,A -85,B 0,C 180,E1 -11595.176,E2 -11595.176} C_VEL
LIN {X 0,Y 390.704,Z 494.76,A -85,B 0,C 180,E1 -11596.342,E2 -11596.342} C_VEL
LIN {X 0,Y 390.183,Z 503.62,A -85,B 0,C 180,E1 -11597.517,E2 -11597.517} C_VEL
LIN {X 0,Y 389.665,Z 513.281,A -85,B 0,C 180,E1 -11599.083,E2 -11599.083} C_VEL
LIN {X 0,Y 389.329,Z 520.991,A -85,B 0,C 180,E1 -11600.65,E2 -11600.65} C_VEL
LIN {X 0,Y 389.313,Z 527.188,A -85,B 0,C 180,E1 -11602.219,E2 -11602.219} C_VEL
LIN {X 0,Y 389.323,Z 532.048,A -85,B 0,C 180,E1 -11603.782,E2 -11603.782} C_VEL
LIN {X 0,Y 389.508,Z 535.734,A -85,B 0,C 180,E1 -11605.343,E2 -11605.343} C_VEL
LIN {X 0,Y 389.538,Z 538.289,A -85,B 0,C 180,E1 -11606.897,E2 -11606.897} C_VEL
LIN {X 0,Y 389.576,Z 539.428,A -85,B 0,C 180,E1 -11607.932,E2 -11607.932} C_VEL
LIN {X 0,Y 389.73,Z 540.138,A -85,B 0,C 180,E1 -11608.967,E2 -11608.967} C_VEL
LIN {X 0,Y 389.885,Z 540.375,A -85,B 0,C 180,E1 -11610,E2 -11610} C_VEL
LIN {X 0,Y 389.813,Z 540.148,A -85,B 0,C 180,E1 -11611.033,E2 -11611.033} C_VEL
LIN {X 0,Y 389.565,Z 539.472,A -85,B 0,C 180,E1 -11612.068,E2 -11612.068} C_VEL
LIN {X 0,Y 389.536,Z 538.372,A -85,B 0,C 180,E1 -11613.103,E2 -11613.103} C_VEL
LIN {X 0,Y 389.498,Z 535.886,A -85,B 0,C 180,E1 -11614.657,E2 -11614.657} C_VEL
LIN {X 0,Y 389.352,Z 532.327,A -85,B 0,C 180,E1 -11616.217,E2 -11616.217} C_VEL
LIN {X 0,Y 389.255,Z 527.652,A -85,B 0,C 180,E1 -11617.782,E2 -11617.782} C_VEL
LIN {X 0,Y 389.335,Z 520.647,A -85,B 0,C 180,E1 -11619.612,E2 -11619.612} C_VEL
LIN {X 0,Y 389.697,Z 513.188,A -85,B 0,C 180,E1 -11621.179,E2 -11621.179} C_VEL
LIN {X 0,Y 390.289,Z 504.11,A -85,B 0,C 180,E1 -11622.744,E2 -11622.744} C_VEL
LIN {X 0,Y 390.946,Z 494.973,A -85,B 0,C 180,E1 -11624.045,E2 -11624.045} C_VEL
LIN {X 0,Y 391.974,Z 484.032,A -85,B 0,C 180,E1 -11625.335,E2 -11625.335} C_VEL
LIN {X 0,Y 393.002,Z 472.106,A -85,B 0,C 180,E1 -11626.493,E2 -11626.493} C_VEL
LIN {X 0,Y 393.045,Z 458.925,A -85,B 0,C 180,E1 -11627.562,E2 -11627.562} C_VEL
LIN {X 0,Y 392.838,Z 446.922,A -85,B 0,C 180,E1 -11628.367,E2 -11628.367} C_VEL
LIN {X 0,Y 391.498,Z 432.955,A -85,B 0,C 180,E1 -11629.175,E2 -11629.175} C_VEL
LIN {X 0,Y 389.583,Z 421.566,A -85,B 0,C 180,E1 -11629.77,E2 -11629.77} C_VEL
LIN {X 0,Y 389.982,Z 408.553,A -85,B 0,C 180,E1 -11633.358,E2 -11633.358} C_VEL
LIN {X 0,Y 390.502,Z 396.731,A -85,B 0,C 180,E1 -11636.74,E2 -11636.74} C_VEL
LIN {X 0,Y 391.292,Z 384.443,A -85,B 0,C 180,E1 -11640.443,E2 -11640.443} C_VEL
LIN {X 0,Y 392.163,Z 374.238,A -85,B 0,C 180,E1 -11643.749,E2 -11643.749} C_VEL
LIN {X 0,Y 393.447,Z 365.345,A -85,B 0,C 180,E1 -11646.866,E2 -11646.866} C_VEL
LIN {X 0,Y 392.913,Z 360.774,A -85,B 0,C 180,E1 -11648.759,E2 -11648.759} C_VEL
LIN {X 0,Y 391.771,Z 354.812,A -85,B 0,C 180,E1 -11651.586,E2 -11651.586} C_VEL
LIN {X 0,Y 390.617,Z 349.61,A -85,B 0,C 180,E1 -11654.563,E2 -11654.563} C_VEL
LIN {X 0,Y 390.071,Z 346.897,A -85,B 0,C 180,E1 -11656.444,E2 -11656.444} C_VEL
LIN {X 0,Y 390.059,Z 346.897,A -85,B 0,C 180,E1 -11659.561,E2 -11659.561} C_VEL
LIN {X 0,Y 390.049,Z 346.898,A -85,B 0,C 180,E1 -11662.449,E2 -11662.449} C_VEL
LIN {X 0,Y 390.087,Z 346.896,A -85,B 0,C 180,E1 -11666.047,E2 -11666.047} C_VEL
LIN {X 0,Y 390.05,Z 346.899,A -85,B 0,C 180,E1 -11669.869,E2 -11669.869} C_VEL
LIN {X 0,Y 390.117,Z 346.89,A -85,B 0,C 180,E1 -11673.232,E2 -11673.232} C_VEL
LIN {X 0,Y 390.11,Z 346.891,A -85,B 0,C 180,E1 -11676.75,E2 -11676.75} C_VEL
LIN {X 0,Y 390.1,Z 346.895,A -85,B 0,C 180,E1 -11679.983,E2 -11679.983} C_VEL
LIN {X 0,Y 392.252,Z 352.246,A -85,B 0,C 180,E1 -11680.51,E2 -11680.51} C_VEL
LIN {X 0,Y 395.797,Z 361.413,A -85,B 0,C 180,E1 -11681.478,E2 -11681.478} C_VEL
LIN {X 0,Y 397.622,Z 367.76,A -85,B 0,C 180,E1 -11682.183,E2 -11682.183} C_VEL
LIN {X 0,Y 396.69,Z 379.672,A -85,B 0,C 180,E1 -11683.319,E2 -11683.319} C_VEL
LIN {X 0,Y 395.665,Z 389.908,A -85,B 0,C 180,E1 -11684.547,E2 -11684.547} C_VEL
LIN {X 0,Y 394.74,Z 398.601,A -85,B 0,C 180,E1 -11685.829,E2 -11685.829} C_VEL
LIN {X 0,Y 393.837,Z 405.791,A -85,B 0,C 180,E1 -11687.111,E2 -11687.111} C_VEL
LIN {X 0,Y 392.957,Z 412.839,A -85,B 0,C 180,E1 -11688.654,E2 -11688.654} C_VEL
LIN {X 0,Y 392.207,Z 418.627,A -85,B 0,C 180,E1 -11690.251,E2 -11690.251} C_VEL
LIN {X 0,Y 391.554,Z 422.88,A -85,B 0,C 180,E1 -11691.744,E2 -11691.744} C_VEL
LIN {X 0,Y 391.219,Z 425.209,A -85,B 0,C 180,E1 -11692.776,E2 -11692.776} C_VEL
LIN {X 0,Y 390.817,Z 427.103,A -85,B 0,C 180,E1 -11693.806,E2 -11693.806} C_VEL
LIN {X 0,Y 390.417,Z 429.51,A -85,B 0,C 180,E1 -11695.871,E2 -11695.871} C_VEL
LIN {X 0,Y 390.295,Z 430.121,A -85,B 0,C 180,E1 -11696.903,E2 -11696.903} C_VEL
LIN {X 0,Y 390.201,Z 430.301,A -85,B 0,C 180,E1 -11697.935,E2 -11697.935} C_VEL
LIN {X 0,Y 390.11,Z 430.085,A -85,B 0,C 180,E1 -11698.968,E2 -11698.968} C_VEL
LIN {X 0,Y 390.056,Z 429.479,A -85,B 0,C 180,E1 -11700,E2 -11700} C_VEL
LIN {X 0,Y 389.925,Z 428.478,A -85,B 0,C 180,E1 -11701.033,E2 -11701.033} C_VEL
LIN {X 0,Y 390.014,Z 427.011,A -85,B 0,C 180,E1 -11702.065,E2 -11702.065} C_VEL
LIN {X 0,Y 390.124,Z 424.038,A -85,B 0,C 180,E1 -11703.615,E2 -11703.615} C_VEL
LIN {X 0,Y 390.272,Z 420.039,A -85,B 0,C 180,E1 -11705.166,E2 -11705.166} C_VEL
LIN {X 0,Y 390.667,Z 414.886,A -85,B 0,C 180,E1 -11706.715,E2 -11706.715} C_VEL
LIN {X 0,Y 391.124,Z 408.46,A -85,B 0,C 180,E1 -11708.265,E2 -11708.265} C_VEL
LIN {X 0,Y 391.549,Z 400.542,A -85,B 0,C 180,E1 -11709.818,E2 -11709.818} C_VEL
LIN {X 0,Y 392.231,Z 390.665,A -85,B 0,C 180,E1 -11711.367,E2 -11711.367} C_VEL
LIN {X 0,Y 392.793,Z 380.573,A -85,B 0,C 180,E1 -11712.661,E2 -11712.661} C_VEL
LIN {X 0,Y 393.424,Z 369.303,A -85,B 0,C 180,E1 -11713.823,E2 -11713.823} C_VEL
LIN {X 0,Y 393.704,Z 360.522,A -85,B 0,C 180,E1 -11714.579,E2 -11714.579} C_VEL
LIN {X 0,Y 390.31,Z 347.64,A -85,B 0,C 180,E1 -11715.605,E2 -11715.605} C_VEL
LIN {X 0,Y 390.175,Z 346.883,A -85,B 0,C 180,E1 -11715.675,E2 -11715.675} C_VEL
LIN {X 0,Y 390.106,Z 346.892,A -85,B 0,C 180,E1 -11718.922,E2 -11718.922} C_VEL
LIN {X 0,Y 390.043,Z 346.898,A -85,B 0,C 180,E1 -11722.234,E2 -11722.234} C_VEL
LIN {X 0,Y 390.122,Z 346.889,A -85,B 0,C 180,E1 -11725.743,E2 -11725.743} C_VEL
LIN {X 0,Y 390.062,Z 346.899,A -85,B 0,C 180,E1 -11729.109,E2 -11729.109} C_VEL
LIN {X 0,Y 390.045,Z 346.9,A -85,B 0,C 180,E1 -11732.721,E2 -11732.721} C_VEL
LIN {X 0,Y 390.059,Z 346.894,A -85,B 0,C 180,E1 -11735.825,E2 -11735.825} C_VEL
LIN {X 0,Y 390.076,Z 346.895,A -85,B 0,C 180,E1 -11739.219,E2 -11739.219} C_VEL
LIN {X 0,Y 390.082,Z 346.896,A -85,B 0,C 180,E1 -11742.38,E2 -11742.38} C_VEL
LIN {X 0,Y 390.059,Z 346.897,A -85,B 0,C 180,E1 -11746.113,E2 -11746.113} C_VEL
LIN {X 0,Y 390.058,Z 346.896,A -85,B 0,C 180,E1 -11749.56,E2 -11749.56} C_VEL
LIN {X 0,Y 390.045,Z 346.9,A -85,B 0,C 180,E1 -11752.449,E2 -11752.449} C_VEL
LIN {X 0,Y 390.069,Z 346.895,A -85,B 0,C 180,E1 -11755.975,E2 -11755.975} C_VEL
LIN {X 0,Y 390.048,Z 346.898,A -85,B 0,C 180,E1 -11759.869,E2 -11759.869} C_VEL
LIN {X 0,Y 390.114,Z 346.89,A -85,B 0,C 180,E1 -11763.232,E2 -11763.232} C_VEL
LIN {X 0,Y 390.107,Z 346.892,A -85,B 0,C 180,E1 -11766.75,E2 -11766.75} C_VEL
LIN {X 0,Y 390.12,Z 346.89,A -85,B 0,C 180,E1 -11769.984,E2 -11769.984} C_VEL
LIN {X 0,Y 390.139,Z 346.885,A -85,B 0,C 180,E1 -11773.248,E2 -11773.248} C_VEL
LIN {X 0,Y 390.195,Z 346.881,A -85,B 0,C 180,E1 -11776.562,E2 -11776.562} C_VEL
LIN {X 0,Y 390.17,Z 346.884,A -85,B 0,C 180,E1 -11779.623,E2 -11779.623} C_VEL
LIN {X 0,Y 390.302,Z 346.867,A -85,B 0,C 180,E1 -11782.759,E2 -11782.759} C_VEL
LIN {X 0,Y 390.226,Z 346.875,A -85,B 0,C 180,E1 -11784.834,E2 -11784.834} C_VEL
LIN {X 0,Y 390.421,Z 346.854,A -85,B 0,C 180,E1 -11787.937,E2 -11787.937} C_VEL
LIN {X 0,Y 390.549,Z 346.839,A -85,B 0,C 180,E1 -11790,E2 -11790} C_VEL
LIN {X 0,Y 390.317,Z 346.864,A -85,B 0,C 180,E1 -11793.097,E2 -11793.097} C_VEL
LIN {X 0,Y 390.325,Z 346.865,A -85,B 0,C 180,E1 -11796.202,E2 -11796.202} C_VEL
LIN {X 0,Y 390.206,Z 346.88,A -85,B 0,C 180,E1 -11799.329,E2 -11799.329} C_VEL
LIN {X 0,Y 390.172,Z 346.882,A -85,B 0,C 180,E1 -11802.483,E2 -11802.483} C_VEL
LIN {X 0,Y 390.141,Z 346.89,A -85,B 0,C 180,E1 -11805.677,E2 -11805.677} C_VEL
LIN {X 0,Y 390.107,Z 346.889,A -85,B 0,C 180,E1 -11808.922,E2 -11808.922} C_VEL
LIN {X 0,Y 390.049,Z 346.898,A -85,B 0,C 180,E1 -11812.234,E2 -11812.234} C_VEL
LIN {X 0,Y 390.12,Z 346.891,A -85,B 0,C 180,E1 -11815.744,E2 -11815.744} C_VEL
LIN {X 0,Y 390.076,Z 346.894,A -85,B 0,C 180,E1 -11818.273,E2 -11818.273} C_VEL
LIN {X 0,Y 389.37,Z 346.984,A -85,B 0,C 180,E1 -11819.134,E2 -11819.134} C_VEL
LIN {X 0,Y 386.492,Z 347.34,A -85,B 0,C 180,E1 -11820.534,E2 -11820.534} C_VEL
LIN {X 0,Y 384.083,Z 347.644,A -85,B 0,C 180,E1 -11821.665,E2 -11821.665} C_VEL
LIN {X 0,Y 383.06,Z 347.767,A -85,B 0,C 180,E1 -11822.54,E2 -11822.54} C_VEL
LIN {X 0,Y 382.981,Z 347.777,A -85,B 0,C 180,E1 -11822.836,E2 -11822.836} C_VEL
LIN {X 0,Y 383.034,Z 347.771,A -85,B 0,C 180,E1 -11826.165,E2 -11826.165} C_VEL
LIN {X 0,Y 383.018,Z 347.774,A -85,B 0,C 180,E1 -11829.958,E2 -11829.958} C_VEL
LIN {X 0,Y 383.067,Z 347.769,A -85,B 0,C 180,E1 -11832.789,E2 -11832.789} C_VEL
LIN {X 0,Y 383.01,Z 347.775,A -85,B 0,C 180,E1 -11835.791,E2 -11835.791} C_VEL
LIN {X 0,Y 382.99,Z 347.778,A -85,B 0,C 180,E1 -11838.796,E2 -11838.796} C_VEL
LIN {X 0,Y 383.002,Z 347.773,A -85,B 0,C 180,E1 -11842.097,E2 -11842.097} C_VEL
LIN {X 0,Y 383.021,Z 347.775,A -85,B 0,C 180,E1 -11845.332,E2 -11845.332} C_VEL
LIN {X 0,Y 382.986,Z 347.78,A -85,B 0,C 180,E1 -11849.082,E2 -11849.082} C_VEL
LIN {X 0,Y 383.06,Z 347.77,A -85,B 0,C 180,E1 -11852.699,E2 -11852.699} C_VEL
LIN {X 0,Y 383.056,Z 347.772,A -85,B 0,C 180,E1 -11855.04,E2 -11855.04} C_VEL
LIN {X 0,Y 382.997,Z 347.777,A -85,B 0,C 180,E1 -11858.469,E2 -11858.469} C_VEL
LIN {X 0,Y 383.067,Z 347.766,A -85,B 0,C 180,E1 -11861.827,E2 -11861.827} C_VEL
LIN {X 0,Y 383.115,Z 347.763,A -85,B 0,C 180,E1 -11865.119,E2 -11865.119} C_VEL
LIN {X 0,Y 383.103,Z 347.766,A -85,B 0,C 180,E1 -11868.358,E2 -11868.358} C_VEL
LIN {X 0,Y 383.309,Z 347.737,A -85,B 0,C 180,E1 -11871.933,E2 -11871.933} C_VEL
LIN {X 0,Y 383.203,Z 347.754,A -85,B 0,C 180,E1 -11874.739,E2 -11874.739} C_VEL
LIN {X 0,Y 383.39,Z 347.726,A -85,B 0,C 180,E1 -11877.899,E2 -11877.899} C_VEL
LIN {X 0,Y 383.523,Z 347.711,A -85,B 0,C 180,E1 -11880,E2 -11880} C_VEL
LIN {X 0,Y 383.256,Z 347.744,A -85,B 0,C 180,E1 -11883.154,E2 -11883.154} C_VEL
LIN {X 0,Y 383.277,Z 347.744,A -85,B 0,C 180,E1 -11886.317,E2 -11886.317} C_VEL
LIN {X 0,Y 383.148,Z 347.757,A -85,B 0,C 180,E1 -11889.502,E2 -11889.502} C_VEL
LIN {X 0,Y 383.141,Z 347.759,A -85,B 0,C 180,E1 -11892.716,E2 -11892.716} C_VEL
LIN {X 0,Y 383.086,Z 347.767,A -85,B 0,C 180,E1 -11895.973,E2 -11895.973} C_VEL
LIN {X 0,Y 383.066,Z 347.767,A -85,B 0,C 180,E1 -11899.284,E2 -11899.284} C_VEL
LIN {X 0,Y 383.042,Z 347.771,A -85,B 0,C 180,E1 -11903.451,E2 -11903.451} C_VEL
LIN {X 0,Y 383.084,Z 347.768,A -85,B 0,C 180,E1 -11906.123,E2 -11906.123} C_VEL
LIN {X 0,Y 383.045,Z 347.771,A -85,B 0,C 180,E1 -11908.493,E2 -11908.493} C_VEL
LIN {X 0,Y 383.014,Z 347.776,A -85,B 0,C 180,E1 -11912.15,E2 -11912.15} C_VEL
LIN {X 0,Y 383.022,Z 347.772,A -85,B 0,C 180,E1 -11914.668,E2 -11914.668} C_VEL
LIN {X 0,Y 383.006,Z 347.778,A -85,B 0,C 180,E1 -11917.904,E2 -11917.904} C_VEL
LIN {X 0,Y 382.988,Z 347.779,A -85,B 0,C 180,E1 -11921.347,E2 -11921.347} C_VEL
LIN {X 0,Y 383.026,Z 347.775,A -85,B 0,C 180,E1 -11924.949,E2 -11924.949} C_VEL
LIN {X 0,Y 383.042,Z 347.819,A -85,B 0,C 180,E1 -11925.503,E2 -11925.503} C_VEL
LIN {X 0,Y 384.9,Z 357.231,A -85,B 0,C 180,E1 -11928.903,E2 -11928.903} C_VEL
LIN {X 0,Y 386.74,Z 366.681,A -85,B 0,C 180,E1 -11932.164,E2 -11932.164} C_VEL
LIN {X 0,Y 386.93,Z 369.769,A -85,B 0,C 180,E1 -11933.173,E2 -11933.173} C_VEL
LIN {X 0,Y 385.505,Z 383.712,A -85,B 0,C 180,E1 -11937.514,E2 -11937.514} C_VEL
LIN {X 0,Y 384.438,Z 396.302,A -85,B 0,C 180,E1 -11941.343,E2 -11941.343} C_VEL
LIN {X 0,Y 383.562,Z 408.782,A -85,B 0,C 180,E1 -11945.075,E2 -11945.075} C_VEL
LIN {X 0,Y 382.895,Z 420.247,A -85,B 0,C 180,E1 -11948.463,E2 -11948.463} C_VEL
LIN {X 0,Y 382.481,Z 431.643,A -85,B 0,C 180,E1 -11951.798,E2 -11951.798} C_VEL
LIN {X 0,Y 383.661,Z 446.337,A -85,B 0,C 180,E1 -11952.377,E2 -11952.377} C_VEL
LIN {X 0,Y 384.561,Z 458.866,A -85,B 0,C 180,E1 -11953.066,E2 -11953.066} C_VEL
LIN {X 0,Y 385.229,Z 471.59,A -85,B 0,C 180,E1 -11953.982,E2 -11953.982} C_VEL
LIN {X 0,Y 384.643,Z 480.71,A -85,B 0,C 180,E1 -11954.772,E2 -11954.772} C_VEL
LIN {X 0,Y 383.84,Z 491.917,A -85,B 0,C 180,E1 -11955.96,E2 -11955.96} C_VEL
LIN {X 0,Y 383.221,Z 502.002,A -85,B 0,C 180,E1 -11957.287,E2 -11957.287} C_VEL
LIN {X 0,Y 382.654,Z 511.755,A -85,B 0,C 180,E1 -11958.881,E2 -11958.881} C_VEL
LIN {X 0,Y 382.3,Z 519.594,A -85,B 0,C 180,E1 -11960.476,E2 -11960.476} C_VEL
LIN {X 0,Y 382.263,Z 525.862,A -85,B 0,C 180,E1 -11962.074,E2 -11962.074} C_VEL
LIN {X 0,Y 382.268,Z 530.786,A -85,B 0,C 180,E1 -11963.667,E2 -11963.667} C_VEL
LIN {X 0,Y 382.48,Z 534.533,A -85,B 0,C 180,E1 -11965.257,E2 -11965.257} C_VEL
LIN {X 0,Y 382.51,Z 537.137,A -85,B 0,C 180,E1 -11966.84,E2 -11966.84} C_VEL
LIN {X 0,Y 382.552,Z 538.297,A -85,B 0,C 180,E1 -11967.894,E2 -11967.894} C_VEL
LIN {X 0,Y 382.712,Z 539.043,A -85,B 0,C 180,E1 -11968.948,E2 -11968.948} C_VEL
LIN {X 0,Y 382.88,Z 539.31,A -85,B 0,C 180,E1 -11970,E2 -11970} C_VEL
LIN {X 0,Y 382.784,Z 539.099,A -85,B 0,C 180,E1 -11971.052,E2 -11971.052} C_VEL
LIN {X 0,Y 382.529,Z 538.437,A -85,B 0,C 180,E1 -11972.106,E2 -11972.106} C_VEL
LIN {X 0,Y 382.492,Z 537.375,A -85,B 0,C 180,E1 -11973.16,E2 -11973.16} C_VEL
LIN {X 0,Y 382.427,Z 534.91,A -85,B 0,C 180,E1 -11974.744,E2 -11974.744} C_VEL
LIN {X 0,Y 382.261,Z 531.382,A -85,B 0,C 180,E1 -11976.333,E2 -11976.333} C_VEL
LIN {X 0,Y 382.199,Z 526.756,A -85,B 0,C 180,E1 -11977.927,E2 -11977.927} C_VEL
LIN {X 0,Y 382.262,Z 519.833,A -85,B 0,C 180,E1 -11979.792,E2 -11979.792} C_VEL
LIN {X 0,Y 382.742,Z 511.092,A -85,B 0,C 180,E1 -11981.653,E2 -11981.653} C_VEL
LIN {X 0,Y 383.348,Z 502.041,A -85,B 0,C 180,E1 -11983.209,E2 -11983.209} C_VEL
LIN {X 0,Y 384.265,Z 492.504,A -85,B 0,C 180,E1 -11984.565,E2 -11984.565} C_VEL
LIN {X 0,Y 385.358,Z 481.396,A -85,B 0,C 180,E1 -11985.877,E2 -11985.877} C_VEL
LIN {X 0,Y 386.125,Z 472.117,A -85,B 0,C 180,E1 -11986.795,E2 -11986.795} C_VEL
LIN {X 0,Y 386.304,Z 459.472,A -85,B 0,C 180,E1 -11987.879,E2 -11987.879} C_VEL
LIN {X 0,Y 386.118,Z 446.001,A -85,B 0,C 180,E1 -11988.828,E2 -11988.828} C_VEL
LIN {X 0,Y 384.696,Z 432.139,A -85,B 0,C 180,E1 -11989.684,E2 -11989.684} C_VEL
LIN {X 0,Y 382.596,Z 419.971,A -85,B 0,C 180,E1 -11990.357,E2 -11990.357} C_VEL
LIN {X 0,Y 383.088,Z 405.833,A -85,B 0,C 180,E1 -11994.38,E2 -11994.38} C_VEL
LIN {X 0,Y 383.676,Z 394.16,A -85,B 0,C 180,E1 -11997.846,E2 -11997.846} C_VEL
LIN {X 0,Y 384.346,Z 384.744,A -85,B 0,C 180,E1 -12000.797,E2 -12000.797} C_VEL
LIN {X 0,Y 385.239,Z 375.686,A -85,B 0,C 180,E1 -12003.809,E2 -12003.809} C_VEL
LIN {X 0,Y 386.542,Z 367.149,A -85,B 0,C 180,E1 -12006.87,E2 -12006.87} C_VEL
LIN {X 0,Y 386.163,Z 363.245,A -85,B 0,C 180,E1 -12008.502,E2 -12008.502} C_VEL
LIN {X 0,Y 384.982,Z 356.913,A -85,B 0,C 180,E1 -12011.542,E2 -12011.542} C_VEL
LIN {X 0,Y 383.882,Z 351.904,A -85,B 0,C 180,E1 -12014.438,E2 -12014.438} C_VEL
LIN {X 0,Y 383.015,Z 347.776,A -85,B 0,C 180,E1 -12017.419,E2 -12017.419} C_VEL
LIN {X 0,Y 383.018,Z 347.774,A -85,B 0,C 180,E1 -12020.413,E2 -12020.413} C_VEL
LIN {X 0,Y 383.03,Z 347.773,A -85,B 0,C 180,E1 -12024.045,E2 -12024.045} C_VEL
LIN {X 0,Y 382.99,Z 347.778,A -85,B 0,C 180,E1 -12027.578,E2 -12027.578} C_VEL
LIN {X 0,Y 382.995,Z 347.776,A -85,B 0,C 180,E1 -12030.3,E2 -12030.3} C_VEL
LIN {X 0,Y 383.06,Z 347.771,A -85,B 0,C 180,E1 -12032.698,E2 -12032.698} C_VEL
LIN {X 0,Y 383.056,Z 347.77,A -85,B 0,C 180,E1 -12035.04,E2 -12035.04} C_VEL
LIN {X 0,Y 382.997,Z 347.778,A -85,B 0,C 180,E1 -12038.469,E2 -12038.469} C_VEL
LIN {X 0,Y 383.062,Z 347.893,A -85,B 0,C 180,E1 -12039.379,E2 -12039.379} C_VEL
LIN {X 0,Y 384.143,Z 350.758,A -85,B 0,C 180,E1 -12039.659,E2 -12039.659} C_VEL
LIN {X 0,Y 388.681,Z 361.52,A -85,B 0,C 180,E1 -12040.869,E2 -12040.869} C_VEL
LIN {X 0,Y 391.232,Z 370.023,A -85,B 0,C 180,E1 -12041.839,E2 -12041.839} C_VEL
LIN {X 0,Y 390.2,Z 381.58,A -85,B 0,C 180,E1 -12042.991,E2 -12042.991} C_VEL
LIN {X 0,Y 389.071,Z 391.886,A -85,B 0,C 180,E1 -12044.279,E2 -12044.279} C_VEL
LIN {X 0,Y 388.093,Z 400.459,A -85,B 0,C 180,E1 -12045.581,E2 -12045.581} C_VEL
LIN {X 0,Y 386.978,Z 408.777,A -85,B 0,C 180,E1 -12047.145,E2 -12047.145} C_VEL
LIN {X 0,Y 386.191,Z 414.439,A -85,B 0,C 180,E1 -12048.452,E2 -12048.452} C_VEL
LIN {X 0,Y 385.46,Z 419.621,A -85,B 0,C 180,E1 -12049.924,E2 -12049.924} C_VEL
LIN {X 0,Y 384.664,Z 424.261,A -85,B 0,C 180,E1 -12051.595,E2 -12051.595} C_VEL
LIN {X 0,Y 384.305,Z 426.557,A -85,B 0,C 180,E1 -12052.645,E2 -12052.645} C_VEL
LIN {X 0,Y 383.877,Z 428.393,A -85,B 0,C 180,E1 -12053.693,E2 -12053.693} C_VEL
LIN {X 0,Y 383.64,Z 429.761,A -85,B 0,C 180,E1 -12054.744,E2 -12054.744} C_VEL
LIN {X 0,Y 383.462,Z 430.725,A -85,B 0,C 180,E1 -12055.796,E2 -12055.796} C_VEL
LIN {X 0,Y 383.31,Z 431.287,A -85,B 0,C 180,E1 -12056.847,E2 -12056.847} C_VEL
LIN {X 0,Y 383.196,Z 431.414,A -85,B 0,C 180,E1 -12057.898,E2 -12057.898} C_VEL
LIN {X 0,Y 383.096,Z 431.157,A -85,B 0,C 180,E1 -12058.949,E2 -12058.949} C_VEL
LIN {X 0,Y 383.038,Z 430.508,A -85,B 0,C 180,E1 -12060,E2 -12060} C_VEL
LIN {X 0,Y 382.9,Z 429.446,A -85,B 0,C 180,E1 -12061.052,E2 -12061.052} C_VEL
LIN {X 0,Y 382.988,Z 427.936,A -85,B 0,C 180,E1 -12062.103,E2 -12062.103} C_VEL
LIN {X 0,Y 382.878,Z 426.05,A -85,B 0,C 180,E1 -12063.157,E2 -12063.157} C_VEL
LIN {X 0,Y 383.339,Z 422.29,A -85,B 0,C 180,E1 -12064.732,E2 -12064.732} C_VEL
LIN {X 0,Y 383.533,Z 417.473,A -85,B 0,C 180,E1 -12066.312,E2 -12066.312} C_VEL
LIN {X 0,Y 383.962,Z 411.404,A -85,B 0,C 180,E1 -12067.89,E2 -12067.89} C_VEL
LIN {X 0,Y 384.425,Z 403.87,A -85,B 0,C 180,E1 -12069.47,E2 -12069.47} C_VEL
LIN {X 0,Y 384.976,Z 394.596,A -85,B 0,C 180,E1 -12071.051,E2 -12071.051} C_VEL
LIN {X 0,Y 385.681,Z 385.09,A -85,B 0,C 180,E1 -12072.363,E2 -12072.363} C_VEL
LIN {X 0,Y 386.25,Z 374.664,A -85,B 0,C 180,E1 -12073.548,E2 -12073.548} C_VEL
LIN {X 0,Y 386.784,Z 362.591,A -85,B 0,C 180,E1 -12074.663,E2 -12074.663} C_VEL
LIN {X 0,Y 383.764,Z 350.366,A -85,B 0,C 180,E1 -12075.671,E2 -12075.671} C_VEL
LIN {X 0,Y 383.13,Z 347.759,A -85,B 0,C 180,E1 -12075.869,E2 -12075.869} C_VEL
LIN {X 0,Y 383.062,Z 347.771,A -85,B 0,C 180,E1 -12079.283,E2 -12079.283} C_VEL
LIN {X 0,Y 383.012,Z 347.775,A -85,B 0,C 180,E1 -12082.664,E2 -12082.664} C_VEL
LIN {X 0,Y 383.083,Z 347.765,A -85,B 0,C 180,E1 -12086.123,E2 -12086.123} C_VEL
LIN {X 0,Y 383.043,Z 347.772,A -85,B 0,C 180,E1 -12088.492,E2 -12088.492} C_VEL
LIN {X 0,Y 383.012,Z 347.774,A -85,B 0,C 180,E1 -12092.149,E2 -12092.149} C_VEL
LIN {X 0,Y 383.02,Z 347.775,A -85,B 0,C 180,E1 -12094.668,E2 -12094.668} C_VEL
LIN {X 0,Y 383.005,Z 347.774,A -85,B 0,C 180,E1 -12097.904,E2 -12097.904} C_VEL
LIN {X 0,Y 383.016,Z 347.775,A -85,B 0,C 180,E1 -12101.343,E2 -12101.343} C_VEL
LIN {X 0,Y 382.999,Z 347.777,A -85,B 0,C 180,E1 -12104.303,E2 -12104.303} C_VEL
LIN {X 0,Y 383.011,Z 347.775,A -85,B 0,C 180,E1 -12107.24,E2 -12107.24} C_VEL
LIN {X 0,Y 383.017,Z 347.775,A -85,B 0,C 180,E1 -12110.413,E2 -12110.413} C_VEL
LIN {X 0,Y 383.026,Z 347.772,A -85,B 0,C 180,E1 -12114.044,E2 -12114.044} C_VEL
LIN {X 0,Y 382.988,Z 347.776,A -85,B 0,C 180,E1 -12117.578,E2 -12117.578} C_VEL
LIN {X 0,Y 382.993,Z 347.78,A -85,B 0,C 180,E1 -12120.3,E2 -12120.3} C_VEL
LIN {X 0,Y 383.081,Z 347.768,A -85,B 0,C 180,E1 -12124.021,E2 -12124.021} C_VEL
LIN {X 0,Y 383.014,Z 347.773,A -85,B 0,C 180,E1 -12127.335,E2 -12127.335} C_VEL
LIN {X 0,Y 383.073,Z 347.767,A -85,B 0,C 180,E1 -12130.717,E2 -12130.717} C_VEL
LIN {X 0,Y 383.082,Z 347.768,A -85,B 0,C 180,E1 -12134.027,E2 -12134.027} C_VEL
LIN {X 0,Y 383.137,Z 347.758,A -85,B 0,C 180,E1 -12137.284,E2 -12137.284} C_VEL
LIN {X 0,Y 383.153,Z 347.759,A -85,B 0,C 180,E1 -12140.498,E2 -12140.498} C_VEL
LIN {X 0,Y 383.281,Z 347.742,A -85,B 0,C 180,E1 -12143.684,E2 -12143.684} C_VEL
LIN {X 0,Y 383.389,Z 347.73,A -85,B 0,C 180,E1 -12147.899,E2 -12147.899} C_VEL
LIN {X 0,Y 383.519,Z 347.715,A -85,B 0,C 180,E1 -12150,E2 -12150} C_VEL
LIN {X 0,Y 383.253,Z 347.744,A -85,B 0,C 180,E1 -12153.154,E2 -12153.154} C_VEL
LIN {X 0,Y 383.281,Z 347.743,A -85,B 0,C 180,E1 -12156.316,E2 -12156.316} C_VEL
LIN {X 0,Y 383.153,Z 347.759,A -85,B 0,C 180,E1 -12159.502,E2 -12159.502} C_VEL
LIN {X 0,Y 383.126,Z 347.762,A -85,B 0,C 180,E1 -12163.536,E2 -12163.536} C_VEL
LIN {X 0,Y 383.096,Z 347.766,A -85,B 0,C 180,E1 -12167.455,E2 -12167.455} C_VEL
LIN {X 0,Y 383.032,Z 347.771,A -85,B 0,C 180,E1 -12170.648,E2 -12170.648} C_VEL
LIN {X 0,Y 383.034,Z 347.774,A -85,B 0,C 180,E1 -12173.808,E2 -12173.808} C_VEL
LIN {X 0,Y 383.081,Z 347.767,A -85,B 0,C 180,E1 -12176.124,E2 -12176.124} C_VEL
LIN {X 0,Y 382.994,Z 347.78,A -85,B 0,C 180,E1 -12179.7,E2 -12179.7} C_VEL
LIN {X 0,Y 382.981,Z 347.777,A -85,B 0,C 180,E1 -12182.836,E2 -12182.836} C_VEL
LIN {X 0,Y 382.322,Z 347.863,A -85,B 0,C 180,E1 -12183.714,E2 -12183.714} C_VEL
LIN {X 0,Y 379.461,Z 348.218,A -85,B 0,C 180,E1 -12185.14,E2 -12185.14} C_VEL
LIN {X 0,Y 377.04,Z 348.517,A -85,B 0,C 180,E1 -12186.294,E2 -12186.294} C_VEL
LIN {X 0,Y 376.013,Z 348.649,A -85,B 0,C 180,E1 -12187.186,E2 -12187.186} C_VEL
LIN {X 0,Y 375.935,Z 348.652,A -85,B 0,C 180,E1 -12187.488,E2 -12187.488} C_VEL
LIN {X 0,Y 376,Z 348.649,A -85,B 0,C 180,E1 -12190.86,E2 -12190.86} C_VEL
LIN {X 0,Y 375.981,Z 348.651,A -85,B 0,C 180,E1 -12193.759,E2 -12193.759} C_VEL
LIN {X 0,Y 375.939,Z 348.657,A -85,B 0,C 180,E1 -12196.81,E2 -12196.81} C_VEL
LIN {X 0,Y 375.965,Z 348.651,A -85,B 0,C 180,E1 -12200.538,E2 -12200.538} C_VEL
LIN {X 0,Y 375.966,Z 348.653,A -85,B 0,C 180,E1 -12203.496,E2 -12203.496} C_VEL
LIN {X 0,Y 375.963,Z 348.652,A -85,B 0,C 180,E1 -12205.889,E2 -12205.889} C_VEL
LIN {X 0,Y 375.968,Z 348.652,A -85,B 0,C 180,E1 -12209.688,E2 -12209.688} C_VEL
LIN {X 0,Y 375.999,Z 348.647,A -85,B 0,C 180,E1 -12212.142,E2 -12212.142} C_VEL
LIN {X 0,Y 376.01,Z 348.648,A -85,B 0,C 180,E1 -12214.539,E2 -12214.539} C_VEL
LIN {X 0,Y 375.967,Z 348.65,A -85,B 0,C 180,E1 -12218.046,E2 -12218.046} C_VEL
LIN {X 0,Y 376.013,Z 348.645,A -85,B 0,C 180,E1 -12221.474,E2 -12221.474} C_VEL
LIN {X 0,Y 376.063,Z 348.642,A -85,B 0,C 180,E1 -12224.833,E2 -12224.833} C_VEL
LIN {X 0,Y 376.055,Z 348.642,A -85,B 0,C 180,E1 -12228.137,E2 -12228.137} C_VEL
LIN {X 0,Y 376.262,Z 348.615,A -85,B 0,C 180,E1 -12231.877,E2 -12231.877} C_VEL
LIN {X 0,Y 376.175,Z 348.63,A -85,B 0,C 180,E1 -12234.64,E2 -12234.64} C_VEL
LIN {X 0,Y 376.356,Z 348.602,A -85,B 0,C 180,E1 -12237.86,E2 -12237.86} C_VEL
LIN {X 0,Y 376.492,Z 348.587,A -85,B 0,C 180,E1 -12240,E2 -12240} C_VEL
LIN {X 0,Y 376.193,Z 348.623,A -85,B 0,C 180,E1 -12243.213,E2 -12243.213} C_VEL
LIN {X 0,Y 376.234,Z 348.621,A -85,B 0,C 180,E1 -12246.435,E2 -12246.435} C_VEL
LIN {X 0,Y 376.118,Z 348.633,A -85,B 0,C 180,E1 -12249.682,E2 -12249.682} C_VEL
LIN {X 0,Y 376.094,Z 348.635,A -85,B 0,C 180,E1 -12253.658,E2 -12253.658} C_VEL
LIN {X 0,Y 376.049,Z 348.641,A -85,B 0,C 180,E1 -12257.608,E2 -12257.608} C_VEL
LIN {X 0,Y 375.983,Z 348.65,A -85,B 0,C 180,E1 -12260.832,E2 -12260.832} C_VEL
LIN {X 0,Y 375.999,Z 348.651,A -85,B 0,C 180,E1 -12264.281,E2 -12264.281} C_VEL
LIN {X 0,Y 376.024,Z 348.645,A -85,B 0,C 180,E1 -12266.652,E2 -12266.652} C_VEL
LIN {X 0,Y 375.975,Z 348.65,A -85,B 0,C 180,E1 -12269.079,E2 -12269.079} C_VEL
LIN {X 0,Y 375.955,Z 348.651,A -85,B 0,C 180,E1 -12272.828,E2 -12272.828} C_VEL
LIN {X 0,Y 375.962,Z 348.653,A -85,B 0,C 180,E1 -12275.415,E2 -12275.415} C_VEL
LIN {X 0,Y 375.98,Z 348.652,A -85,B 0,C 180,E1 -12278.271,E2 -12278.271} C_VEL
LIN {X 0,Y 375.938,Z 348.658,A -85,B 0,C 180,E1 -12281.601,E2 -12281.601} C_VEL
LIN {X 0,Y 376.013,Z 348.805,A -85,B 0,C 180,E1 -12285.256,E2 -12285.256} C_VEL
LIN {X 0,Y 377.883,Z 358.373,A -85,B 0,C 180,E1 -12288.778,E2 -12288.778} C_VEL
LIN {X 0,Y 379.544,Z 366.812,A -85,B 0,C 180,E1 -12291.751,E2 -12291.751} C_VEL
LIN {X 0,Y 379.935,Z 369.571,A -85,B 0,C 180,E1 -12292.694,E2 -12292.694} C_VEL
LIN {X 0,Y 379.034,Z 378.535,A -85,B 0,C 180,E1 -12295.561,E2 -12295.561} C_VEL
LIN {X 0,Y 378.08,Z 388.729,A -85,B 0,C 180,E1 -12298.769,E2 -12298.769} C_VEL
LIN {X 0,Y 377.13,Z 399.945,A -85,B 0,C 180,E1 -12302.232,E2 -12302.232} C_VEL
LIN {X 0,Y 376.249,Z 413.112,A -85,B 0,C 180,E1 -12306.246,E2 -12306.246} C_VEL
LIN {X 0,Y 375.57,Z 426.66,A -85,B 0,C 180,E1 -12310.316,E2 -12310.316} C_VEL
LIN {X 0,Y 375.409,Z 430.81,A -85,B 0,C 180,E1 -12311.557,E2 -12311.557} C_VEL
LIN {X 0,Y 376.466,Z 444.578,A -85,B 0,C 180,E1 -12312.106,E2 -12312.106} C_VEL
LIN {X 0,Y 377.474,Z 458.329,A -85,B 0,C 180,E1 -12312.878,E2 -12312.878} C_VEL
LIN {X 0,Y 378.144,Z 470.966,A -85,B 0,C 180,E1 -12313.812,E2 -12313.812} C_VEL
LIN {X 0,Y 377.806,Z 478.684,A -85,B 0,C 180,E1 -12314.49,E2 -12314.49} C_VEL
LIN {X 0,Y 376.886,Z 490.02,A -85,B 0,C 180,E1 -12315.695,E2 -12315.695} C_VEL
LIN {X 0,Y 376.247,Z 500.302,A -85,B 0,C 180,E1 -12317.047,E2 -12317.047} C_VEL
LIN {X 0,Y 375.596,Z 510.157,A -85,B 0,C 180,E1 -12318.669,E2 -12318.669} C_VEL
LIN {X 0,Y 375.278,Z 518.129,A -85,B 0,C 180,E1 -12320.297,E2 -12320.297} C_VEL
LIN {X 0,Y 375.209,Z 524.49,A -85,B 0,C 180,E1 -12321.924,E2 -12321.924} C_VEL
LIN {X 0,Y 375.219,Z 529.488,A -85,B 0,C 180,E1 -12323.547,E2 -12323.547} C_VEL
LIN {X 0,Y 375.449,Z 533.304,A -85,B 0,C 180,E1 -12325.168,E2 -12325.168} C_VEL
LIN {X 0,Y 375.483,Z 535.967,A -85,B 0,C 180,E1 -12326.781,E2 -12326.781} C_VEL
LIN {X 0,Y 375.53,Z 537.152,A -85,B 0,C 180,E1 -12327.855,E2 -12327.855} C_VEL
LIN {X 0,Y 375.693,Z 537.924,A -85,B 0,C 180,E1 -12328.928,E2 -12328.928} C_VEL
LIN {X 0,Y 375.872,Z 538.242,A -85,B 0,C 180,E1 -12330,E2 -12330} C_VEL
LIN {X 0,Y 375.754,Z 538.045,A -85,B 0,C 180,E1 -12331.072,E2 -12331.072} C_VEL
LIN {X 0,Y 375.492,Z 537.402,A -85,B 0,C 180,E1 -12332.145,E2 -12332.145} C_VEL
LIN {X 0,Y 375.449,Z 536.364,A -85,B 0,C 180,E1 -12333.219,E2 -12333.219} C_VEL
LIN {X 0,Y 375.448,Z 534.866,A -85,B 0,C 180,E1 -12334.294,E2 -12334.294} C_VEL
LIN {X 0,Y 375.213,Z 531.738,A -85,B 0,C 180,E1 -12335.913,E2 -12335.913} C_VEL
LIN {X 0,Y 375.086,Z 527.538,A -85,B 0,C 180,E1 -12337.537,E2 -12337.537} C_VEL
LIN {X 0,Y 375.137,Z 521.164,A -85,B 0,C 180,E1 -12339.435,E2 -12339.435} C_VEL
LIN {X 0,Y 375.456,Z 514.346,A -85,B 0,C 180,E1 -12341.062,E2 -12341.062} C_VEL
LIN {X 0,Y 376.023,Z 506.069,A -85,B 0,C 180,E1 -12342.686,E2 -12342.686} C_VEL
LIN {X 0,Y 376.667,Z 497.812,A -85,B 0,C 180,E1 -12344.038,E2 -12344.038} C_VEL
LIN {X 0,Y 377.889,Z 486.949,A -85,B 0,C 180,E1 -12345.507,E2 -12345.507} C_VEL
LIN {X 0,Y 379.223,Z 474.971,A -85,B 0,C 180,E1 -12346.832,E2 -12346.832} C_VEL
LIN {X 0,Y 379.423,Z 463.363,A -85,B 0,C 180,E1 -12347.935,E2 -12347.935} C_VEL
LIN {X 0,Y 379.626,Z 450.295,A -85,B 0,C 180,E1 -12348.954,E2 -12348.954} C_VEL
LIN {X 0,Y 378.749,Z 437.293,A -85,B 0,C 180,E1 -12349.843,E2 -12349.843} C_VEL
LIN {X 0,Y 376.324,Z 422.152,A -85,B 0,C 180,E1 -12350.773,E2 -12350.773} C_VEL
LIN {X 0,Y 375.569,Z 418.271,A -85,B 0,C 180,E1 -12351.014,E2 -12351.014} C_VEL
LIN {X 0,Y 376.112,Z 405.125,A -85,B 0,C 180,E1 -12354.862,E2 -12354.862} C_VEL
LIN {X 0,Y 376.729,Z 393.966,A -85,B 0,C 180,E1 -12358.287,E2 -12358.287} C_VEL
LIN {X 0,Y 377.483,Z 384.288,A -85,B 0,C 180,E1 -12361.42,E2 -12361.42} C_VEL
LIN {X 0,Y 378.493,Z 375.392,A -85,B 0,C 180,E1 -12364.495,E2 -12364.495} C_VEL
LIN {X 0,Y 379.572,Z 369.165,A -85,B 0,C 180,E1 -12366.796,E2 -12366.796} C_VEL
LIN {X 0,Y 379.401,Z 365.659,A -85,B 0,C 180,E1 -12368.267,E2 -12368.267} C_VEL
LIN {X 0,Y 378.309,Z 359.507,A -85,B 0,C 180,E1 -12371.232,E2 -12371.232} C_VEL
LIN {X 0,Y 377.175,Z 354.337,A -85,B 0,C 180,E1 -12374.218,E2 -12374.218} C_VEL
LIN {X 0,Y 376.12,Z 349.474,A -85,B 0,C 180,E1 -12377.725,E2 -12377.725} C_VEL
LIN {X 0,Y 375.967,Z 348.656,A -85,B 0,C 180,E1 -12378.586,E2 -12378.586} C_VEL
LIN {X 0,Y 375.969,Z 348.652,A -85,B 0,C 180,E1 -12381.912,E2 -12381.912} C_VEL
LIN {X 0,Y 375.983,Z 348.65,A -85,B 0,C 180,E1 -12385.333,E2 -12385.333} C_VEL
LIN {X 0,Y 375.961,Z 348.652,A -85,B 0,C 180,E1 -12388.438,E2 -12388.438} C_VEL
LIN {X 0,Y 375.999,Z 348.647,A -85,B 0,C 180,E1 -12392.141,E2 -12392.141} C_VEL
LIN {X 0,Y 376.01,Z 348.649,A -85,B 0,C 180,E1 -12394.539,E2 -12394.539} C_VEL
LIN {X 0,Y 375.967,Z 348.655,A -85,B 0,C 180,E1 -12398.046,E2 -12398.046} C_VEL
LIN {X 0,Y 375.966,Z 348.667,A -85,B 0,C 180,E1 -12398.693,E2 -12398.693} C_VEL
LIN {X 0,Y 376.645,Z 350.877,A -85,B 0,C 180,E1 -12398.904,E2 -12398.904} C_VEL
LIN {X 0,Y 381.216,Z 360.801,A -85,B 0,C 180,E1 -12400.09,E2 -12400.09} C_VEL
LIN {X 0,Y 383.822,Z 368.362,A -85,B 0,C 180,E1 -12401.003,E2 -12401.003} C_VEL
LIN {X 0,Y 384.848,Z 372.276,A -85,B 0,C 180,E1 -12401.485,E2 -12401.485} C_VEL
LIN {X 0,Y 383.912,Z 382.202,A -85,B 0,C 180,E1 -12402.492,E2 -12402.492} C_VEL
LIN {X 0,Y 382.752,Z 392.184,A -85,B 0,C 180,E1 -12403.739,E2 -12403.739} C_VEL
LIN {X 0,Y 381.676,Z 400.816,A -85,B 0,C 180,E1 -12405.061,E2 -12405.061} C_VEL
LIN {X 0,Y 380.446,Z 409.268,A -85,B 0,C 180,E1 -12406.649,E2 -12406.649} C_VEL
LIN {X 0,Y 379.423,Z 416.066,A -85,B 0,C 180,E1 -12408.243,E2 -12408.243} C_VEL
LIN {X 0,Y 378.541,Z 421.896,A -85,B 0,C 180,E1 -12409.984,E2 -12409.984} C_VEL
LIN {X 0,Y 377.79,Z 425.71,A -85,B 0,C 180,E1 -12411.441,E2 -12411.441} C_VEL
LIN {X 0,Y 377.399,Z 427.936,A -85,B 0,C 180,E1 -12412.51,E2 -12412.51} C_VEL
LIN {X 0,Y 376.941,Z 429.694,A -85,B 0,C 180,E1 -12413.577,E2 -12413.577} C_VEL
LIN {X 0,Y 376.503,Z 431.938,A -85,B 0,C 180,E1 -12415.718,E2 -12415.718} C_VEL
LIN {X 0,Y 376.323,Z 432.441,A -85,B 0,C 180,E1 -12416.788,E2 -12416.788} C_VEL
LIN {X 0,Y 376.189,Z 432.53,A -85,B 0,C 180,E1 -12417.859,E2 -12417.859} C_VEL
LIN {X 0,Y 376.08,Z 432.229,A -85,B 0,C 180,E1 -12418.929,E2 -12418.929} C_VEL
LIN {X 0,Y 376.018,Z 431.531,A -85,B 0,C 180,E1 -12420,E2 -12420} C_VEL
LIN {X 0,Y 375.875,Z 430.406,A -85,B 0,C 180,E1 -12421.071,E2 -12421.071} C_VEL
LIN {X 0,Y 375.963,Z 428.854,A -85,B 0,C 180,E1 -12422.142,E2 -12422.142} C_VEL
LIN {X 0,Y 375.843,Z 426.919,A -85,B 0,C 180,E1 -12423.216,E2 -12423.216} C_VEL
LIN {X 0,Y 376.297,Z 423.082,A -85,B 0,C 180,E1 -12424.821,E2 -12424.821} C_VEL
LIN {X 0,Y 376.511,Z 418.178,A -85,B 0,C 180,E1 -12426.43,E2 -12426.43} C_VEL
LIN {X 0,Y 376.955,Z 412.001,A -85,B 0,C 180,E1 -12428.038,E2 -12428.038} C_VEL
LIN {X 0,Y 377.441,Z 404.371,A -85,B 0,C 180,E1 -12429.647,E2 -12429.647} C_VEL
LIN {X 0,Y 378.035,Z 394.975,A -85,B 0,C 180,E1 -12431.256,E2 -12431.256} C_VEL
LIN {X 0,Y 378.742,Z 384.227,A -85,B 0,C 180,E1 -12432.73,E2 -12432.73} C_VEL
LIN {X 0,Y 379.403,Z 373.439,A -85,B 0,C 180,E1 -12433.934,E2 -12433.934} C_VEL
LIN {X 0,Y 379.8,Z 363.766,A -85,B 0,C 180,E1 -12434.824,E2 -12434.824} C_VEL
LIN {X 0,Y 376.639,Z 350.924,A -85,B 0,C 180,E1 -12435.906,E2 -12435.906} C_VEL
LIN {X 0,Y 376.067,Z 348.638,A -85,B 0,C 180,E1 -12436.105,E2 -12436.105} C_VEL
LIN {X 0,Y 375.999,Z 348.648,A -85,B 0,C 180,E1 -12439.66,E2 -12439.66} C_VEL
LIN {X 0,Y 375.998,Z 348.648,A -85,B 0,C 180,E1 -12443.667,E2 -12443.667} C_VEL
LIN {X 0,Y 376.022,Z 348.647,A -85,B 0,C 180,E1 -12446.652,E2 -12446.652} C_VEL
LIN {X 0,Y 375.973,Z 348.654,A -85,B 0,C 180,E1 -12449.079,E2 -12449.079} C_VEL
LIN {X 0,Y 375.951,Z 348.656,A -85,B 0,C 180,E1 -12452.828,E2 -12452.828} C_VEL
LIN {X 0,Y 375.96,Z 348.652,A -85,B 0,C 180,E1 -12455.415,E2 -12455.415} C_VEL
LIN {X 0,Y 375.98,Z 348.65,A -85,B 0,C 180,E1 -12458.271,E2 -12458.271} C_VEL
LIN {X 0,Y 375.962,Z 348.652,A -85,B 0,C 180,E1 -12461.605,E2 -12461.605} C_VEL
LIN {X 0,Y 375.956,Z 348.654,A -85,B 0,C 180,E1 -12465.264,E2 -12465.264} C_VEL
LIN {X 0,Y 375.942,Z 348.656,A -85,B 0,C 180,E1 -12469.133,E2 -12469.133} C_VEL
LIN {X 0,Y 375.965,Z 348.651,A -85,B 0,C 180,E1 -12471.911,E2 -12471.911} C_VEL
LIN {X 0,Y 375.981,Z 348.649,A -85,B 0,C 180,E1 -12475.332,E2 -12475.332} C_VEL
LIN {X 0,Y 375.959,Z 348.656,A -85,B 0,C 180,E1 -12478.438,E2 -12478.438} C_VEL
LIN {X 0,Y 375.984,Z 348.652,A -85,B 0,C 180,E1 -12482.14,E2 -12482.14} C_VEL
LIN {X 0,Y 376.007,Z 348.65,A -85,B 0,C 180,E1 -12484.539,E2 -12484.539} C_VEL
LIN {X 0,Y 375.972,Z 348.653,A -85,B 0,C 180,E1 -12488.046,E2 -12488.046} C_VEL
LIN {X 0,Y 376.031,Z 348.642,A -85,B 0,C 180,E1 -12491.474,E2 -12491.474} C_VEL
LIN {X 0,Y 376.059,Z 348.64,A -85,B 0,C 180,E1 -12494.833,E2 -12494.833} C_VEL
LIN {X 0,Y 376.051,Z 348.644,A -85,B 0,C 180,E1 -12498.137,E2 -12498.137} C_VEL
LIN {X 0,Y 376.219,Z 348.623,A -85,B 0,C 180,E1 -12501.919,E2 -12501.919} C_VEL
LIN {X 0,Y 376.171,Z 348.627,A -85,B 0,C 180,E1 -12504.64,E2 -12504.64} C_VEL
LIN {X 0,Y 376.355,Z 348.606,A -85,B 0,C 180,E1 -12507.86,E2 -12507.86} C_VEL
LIN {X 0,Y 376.488,Z 348.591,A -85,B 0,C 180,E1 -12510,E2 -12510} C_VEL
LIN {X 0,Y 376.191,Z 348.623,A -85,B 0,C 180,E1 -12513.213,E2 -12513.213} C_VEL
LIN {X 0,Y 376.24,Z 348.619,A -85,B 0,C 180,E1 -12516.435,E2 -12516.435} C_VEL
LIN {X 0,Y 376.12,Z 348.635,A -85,B 0,C 180,E1 -12519.682,E2 -12519.682} C_VEL
LIN {X 0,Y 376.09,Z 348.639,A -85,B 0,C 180,E1 -12523.658,E2 -12523.658} C_VEL
LIN {X 0,Y 376.045,Z 348.646,A -85,B 0,C 180,E1 -12527.608,E2 -12527.608} C_VEL
LIN {X 0,Y 375.979,Z 348.649,A -85,B 0,C 180,E1 -12530.832,E2 -12530.832} C_VEL
LIN {X 0,Y 375.995,Z 348.648,A -85,B 0,C 180,E1 -12534.282,E2 -12534.282} C_VEL
LIN {X 0,Y 376.021,Z 348.645,A -85,B 0,C 180,E1 -12536.652,E2 -12536.652} C_VEL
LIN {X 0,Y 375.966,Z 348.651,A -85,B 0,C 180,E1 -12540.313,E2 -12540.313} C_VEL
LIN {X 0,Y 375.961,Z 348.651,A -85,B 0,C 180,E1 -12544.112,E2 -12544.112} C_VEL
LIN {X 0,Y 375.935,Z 348.652,A -85,B 0,C 180,E1 -12547.488,E2 -12547.488} C_VEL
LIN {X 0,Y 375.295,Z 348.735,A -85,B 0,C 180,E1 -12548.382,E2 -12548.382} C_VEL
LIN {X 0,Y 372.48,Z 349.087,A -85,B 0,C 180,E1 -12549.838,E2 -12549.838} C_VEL
LIN {X 0,Y 370.074,Z 349.388,A -85,B 0,C 180,E1 -12551.014,E2 -12551.014} C_VEL
LIN {X 0,Y 369.024,Z 349.517,A -85,B 0,C 180,E1 -12551.924,E2 -12551.924} C_VEL
LIN {X 0,Y 368.93,Z 349.527,A -85,B 0,C 180,E1 -12552.232,E2 -12552.232} C_VEL
LIN {X 0,Y 368.926,Z 349.531,A -85,B 0,C 180,E1 -12555.183,E2 -12555.183} C_VEL
LIN {X 0,Y 368.885,Z 349.533,A -85,B 0,C 180,E1 -12558.178,E2 -12558.178} C_VEL
LIN {X 0,Y 368.911,Z 349.533,A -85,B 0,C 180,E1 -12561.36,E2 -12561.36} C_VEL
LIN {X 0,Y 368.939,Z 349.53,A -85,B 0,C 180,E1 -12565.147,E2 -12565.147} C_VEL
LIN {X 0,Y 368.932,Z 349.531,A -85,B 0,C 180,E1 -12569.047,E2 -12569.047} C_VEL
LIN {X 0,Y 368.983,Z 349.522,A -85,B 0,C 180,E1 -12571.564,E2 -12571.564} C_VEL
LIN {X 0,Y 369.004,Z 349.518,A -85,B 0,C 180,E1 -12574.02,E2 -12574.02} C_VEL
LIN {X 0,Y 368.936,Z 349.526,A -85,B 0,C 180,E1 -12577.605,E2 -12577.605} C_VEL
LIN {X 0,Y 368.962,Z 349.526,A -85,B 0,C 180,E1 -12581.106,E2 -12581.106} C_VEL
LIN {X 0,Y 369.002,Z 349.522,A -85,B 0,C 180,E1 -12584.536,E2 -12584.536} C_VEL
LIN {X 0,Y 369.01,Z 349.518,A -85,B 0,C 180,E1 -12587.907,E2 -12587.907} C_VEL
LIN {X 0,Y 369.234,Z 349.49,A -85,B 0,C 180,E1 -12591.8,E2 -12591.8} C_VEL
LIN {X 0,Y 369.149,Z 349.504,A -85,B 0,C 180,E1 -12594.538,E2 -12594.538} C_VEL
LIN {X 0,Y 369.321,Z 349.478,A -85,B 0,C 180,E1 -12597.819,E2 -12597.819} C_VEL
LIN {X 0,Y 369.462,Z 349.462,A -85,B 0,C 180,E1 -12600,E2 -12600} C_VEL
LIN {X 0,Y 369.324,Z 349.482,A -85,B 0,C 180,E1 -12602.181,E2 -12602.181} C_VEL
LIN {X 0,Y 369.192,Z 349.499,A -85,B 0,C 180,E1 -12606.559,E2 -12606.559} C_VEL
LIN {X 0,Y 369.068,Z 349.512,A -85,B 0,C 180,E1 -12609.868,E2 -12609.868} C_VEL
LIN {X 0,Y 369.042,Z 349.514,A -85,B 0,C 180,E1 -12613.772,E2 -12613.772} C_VEL
LIN {X 0,Y 369.006,Z 349.52,A -85,B 0,C 180,E1 -12617.768,E2 -12617.768} C_VEL
LIN {X 0,Y 368.934,Z 349.527,A -85,B 0,C 180,E1 -12621.22,E2 -12621.22} C_VEL
LIN {X 0,Y 368.962,Z 349.524,A -85,B 0,C 180,E1 -12624.775,E2 -12624.775} C_VEL
LIN {X 0,Y 368.973,Z 349.522,A -85,B 0,C 180,E1 -12627.203,E2 -12627.203} C_VEL
LIN {X 0,Y 368.923,Z 349.531,A -85,B 0,C 180,E1 -12629.69,E2 -12629.69} C_VEL
LIN {X 0,Y 368.903,Z 349.53,A -85,B 0,C 180,E1 -12633.044,E2 -12633.044} C_VEL
LIN {X 0,Y 368.922,Z 349.531,A -85,B 0,C 180,E1 -12636.197,E2 -12636.197} C_VEL
LIN {X 0,Y 368.908,Z 349.53,A -85,B 0,C 180,E1 -12638.953,E2 -12638.953} C_VEL
LIN {X 0,Y 368.885,Z 349.537,A -85,B 0,C 180,E1 -12642.009,E2 -12642.009} C_VEL
LIN {X 0,Y 368.985,Z 349.626,A -85,B 0,C 180,E1 -12644.95,E2 -12644.95} C_VEL
LIN {X 0,Y 370.939,Z 359.795,A -85,B 0,C 180,E1 -12648.767,E2 -12648.767} C_VEL
LIN {X 0,Y 372.702,Z 368.753,A -85,B 0,C 180,E1 -12651.972,E2 -12651.972} C_VEL
LIN {X 0,Y 372.923,Z 371.488,A -85,B 0,C 180,E1 -12652.91,E2 -12652.91} C_VEL
LIN {X 0,Y 371.626,Z 383.274,A -85,B 0,C 180,E1 -12656.74,E2 -12656.74} C_VEL
LIN {X 0,Y 370.521,Z 394.932,A -85,B 0,C 180,E1 -12660.451,E2 -12660.451} C_VEL
LIN {X 0,Y 369.597,Z 406.462,A -85,B 0,C 180,E1 -12664.065,E2 -12664.065} C_VEL
LIN {X 0,Y 368.87,Z 417.867,A -85,B 0,C 180,E1 -12667.601,E2 -12667.601} C_VEL
LIN {X 0,Y 368.355,Z 429.991,A -85,B 0,C 180,E1 -12671.315,E2 -12671.315} C_VEL
LIN {X 0,Y 369.418,Z 444.459,A -85,B 0,C 180,E1 -12671.912,E2 -12671.912} C_VEL
LIN {X 0,Y 370.407,Z 457.702,A -85,B 0,C 180,E1 -12672.683,E2 -12672.683} C_VEL
LIN {X 0,Y 371.025,Z 470.246,A -85,B 0,C 180,E1 -12673.634,E2 -12673.634} C_VEL
LIN {X 0,Y 370.897,Z 476.522,A -85,B 0,C 180,E1 -12674.193,E2 -12674.193} C_VEL
LIN {X 0,Y 370.051,Z 486.945,A -85,B 0,C 180,E1 -12675.284,E2 -12675.284} C_VEL
LIN {X 0,Y 369.264,Z 497.015,A -85,B 0,C 180,E1 -12676.584,E2 -12676.584} C_VEL
LIN {X 0,Y 368.743,Z 505.421,A -85,B 0,C 180,E1 -12677.898,E2 -12677.898} C_VEL
LIN {X 0,Y 368.316,Z 514.123,A -85,B 0,C 180,E1 -12679.556,E2 -12679.556} C_VEL
LIN {X 0,Y 368.171,Z 521.072,A -85,B 0,C 180,E1 -12681.216,E2 -12681.216} C_VEL
LIN {X 0,Y 368.165,Z 527.106,A -85,B 0,C 180,E1 -12683.048,E2 -12683.048} C_VEL
LIN {X 0,Y 368.325,Z 530.869,A -85,B 0,C 180,E1 -12684.525,E2 -12684.525} C_VEL
LIN {X 0,Y 368.443,Z 533.08,A -85,B 0,C 180,E1 -12685.624,E2 -12685.624} C_VEL
LIN {X 0,Y 368.457,Z 534.778,A -85,B 0,C 180,E1 -12686.72,E2 -12686.72} C_VEL
LIN {X 0,Y 368.508,Z 535.991,A -85,B 0,C 180,E1 -12687.814,E2 -12687.814} C_VEL
LIN {X 0,Y 368.674,Z 536.787,A -85,B 0,C 180,E1 -12688.908,E2 -12688.908} C_VEL
LIN {X 0,Y 368.863,Z 537.155,A -85,B 0,C 180,E1 -12690,E2 -12690} C_VEL
LIN {X 0,Y 368.725,Z 536.99,A -85,B 0,C 180,E1 -12691.092,E2 -12691.092} C_VEL
LIN {X 0,Y 368.455,Z 536.366,A -85,B 0,C 180,E1 -12692.186,E2 -12692.186} C_VEL
LIN {X 0,Y 368.403,Z 535.349,A -85,B 0,C 180,E1 -12693.281,E2 -12693.281} C_VEL
LIN {X 0,Y 368.368,Z 533.897,A -85,B 0,C 180,E1 -12694.377,E2 -12694.377} C_VEL
LIN {X 0,Y 368.144,Z 530.811,A -85,B 0,C 180,E1 -12696.027,E2 -12696.027} C_VEL
LIN {X 0,Y 368.012,Z 526.666,A -85,B 0,C 180,E1 -12697.682,E2 -12697.682} C_VEL
LIN {X 0,Y 368.077,Z 520.381,A -85,B 0,C 180,E1 -12699.618,E2 -12699.618} C_VEL
LIN {X 0,Y 368.53,Z 512.414,A -85,B 0,C 180,E1 -12701.551,E2 -12701.551} C_VEL
LIN {X 0,Y 369.188,Z 503.996,A -85,B 0,C 180,E1 -12703.205,E2 -12703.205} C_VEL
LIN {X 0,Y 370.002,Z 495.611,A -85,B 0,C 180,E1 -12704.577,E2 -12704.577} C_VEL
LIN {X 0,Y 371.287,Z 484.602,A -85,B 0,C 180,E1 -12706.071,E2 -12706.071} C_VEL
LIN {X 0,Y 372.392,Z 475.071,A -85,B 0,C 180,E1 -12707.151,E2 -12707.151} C_VEL
LIN {X 0,Y 372.807,Z 462.359,A -85,B 0,C 180,E1 -12708.407,E2 -12708.407} C_VEL
LIN {X 0,Y 372.981,Z 448.935,A -85,B 0,C 180,E1 -12709.495,E2 -12709.495} C_VEL
LIN {X 0,Y 371.989,Z 436.147,A -85,B 0,C 180,E1 -12710.422,E2 -12710.422} C_VEL
LIN {X 0,Y 369.443,Z 420.806,A -85,B 0,C 180,E1 -12711.435,E2 -12711.435} C_VEL
LIN {X 0,Y 368.557,Z 416.586,A -85,B 0,C 180,E1 -12711.708,E2 -12711.708} C_VEL
LIN {X 0,Y 369.148,Z 404.479,A -85,B 0,C 180,E1 -12715.364,E2 -12715.364} C_VEL
LIN {X 0,Y 369.9,Z 392.783,A -85,B 0,C 180,E1 -12719.074,E2 -12719.074} C_VEL
LIN {X 0,Y 370.938,Z 382.114,A -85,B 0,C 180,E1 -12722.682,E2 -12722.682} C_VEL
LIN {X 0,Y 372.496,Z 371.83,A -85,B 0,C 180,E1 -12726.464,E2 -12726.464} C_VEL
LIN {X 0,Y 372.772,Z 368.925,A -85,B 0,C 180,E1 -12727.642,E2 -12727.642} C_VEL
LIN {X 0,Y 371.933,Z 363.944,A -85,B 0,C 180,E1 -12729.976,E2 -12729.976} C_VEL
LIN {X 0,Y 370.856,Z 358.352,A -85,B 0,C 180,E1 -12733.018,E2 -12733.018} C_VEL
LIN {X 0,Y 369.755,Z 353.505,A -85,B 0,C 180,E1 -12736.243,E2 -12736.243} C_VEL
LIN {X 0,Y 368.915,Z 349.532,A -85,B 0,C 180,E1 -12739.643,E2 -12739.643} C_VEL
LIN {X 0,Y 368.906,Z 349.534,A -85,B 0,C 180,E1 -12743.144,E2 -12743.144} C_VEL
LIN {X 0,Y 368.901,Z 349.534,A -85,B 0,C 180,E1 -12746.462,E2 -12746.462} C_VEL
LIN {X 0,Y 368.932,Z 349.528,A -85,B 0,C 180,E1 -12749.046,E2 -12749.046} C_VEL
LIN {X 0,Y 368.983,Z 349.522,A -85,B 0,C 180,E1 -12751.564,E2 -12751.564} C_VEL
LIN {X 0,Y 369.003,Z 349.52,A -85,B 0,C 180,E1 -12754.02,E2 -12754.02} C_VEL
LIN {X 0,Y 368.936,Z 349.532,A -85,B 0,C 180,E1 -12757.605,E2 -12757.605} C_VEL
LIN {X 0,Y 368.961,Z 349.714,A -85,B 0,C 180,E1 -12757.976,E2 -12757.976} C_VEL
LIN {X 0,Y 369.47,Z 351.476,A -85,B 0,C 180,E1 -12758.155,E2 -12758.155} C_VEL
LIN {X 0,Y 373.595,Z 359.894,A -85,B 0,C 180,E1 -12759.225,E2 -12759.225} C_VEL
LIN {X 0,Y 377.509,Z 370.436,A -85,B 0,C 180,E1 -12760.571,E2 -12760.571} C_VEL
LIN {X 0,Y 378.548,Z 374.74,A -85,B 0,C 180,E1 -12761.115,E2 -12761.115} C_VEL
LIN {X 0,Y 377.479,Z 384.688,A -85,B 0,C 180,E1 -12762.184,E2 -12762.184} C_VEL
LIN {X 0,Y 376.229,Z 394.362,A -85,B 0,C 180,E1 -12763.449,E2 -12763.449} C_VEL
LIN {X 0,Y 375.081,Z 402.85,A -85,B 0,C 180,E1 -12764.792,E2 -12764.792} C_VEL
LIN {X 0,Y 373.792,Z 411.119,A -85,B 0,C 180,E1 -12766.407,E2 -12766.407} C_VEL
LIN {X 0,Y 372.682,Z 417.74,A -85,B 0,C 180,E1 -12768.028,E2 -12768.028} C_VEL
LIN {X 0,Y 371.681,Z 423.665,A -85,B 0,C 180,E1 -12769.878,E2 -12769.878} C_VEL
LIN {X 0,Y 370.757,Z 428.285,A -85,B 0,C 180,E1 -12771.826,E2 -12771.826} C_VEL
LIN {X 0,Y 370.041,Z 431.035,A -85,B 0,C 180,E1 -12773.456,E2 -12773.456} C_VEL
LIN {X 0,Y 369.75,Z 432.307,A -85,B 0,C 180,E1 -12774.546,E2 -12774.546} C_VEL
LIN {X 0,Y 369.54,Z 433.172,A -85,B 0,C 180,E1 -12775.637,E2 -12775.637} C_VEL
LIN {X 0,Y 369.182,Z 433.642,A -85,B 0,C 180,E1 -12777.818,E2 -12777.818} C_VEL
LIN {X 0,Y 369.064,Z 433.298,A -85,B 0,C 180,E1 -12778.909,E2 -12778.909} C_VEL
LIN {X 0,Y 368.998,Z 432.538,A -85,B 0,C 180,E1 -12780,E2 -12780} C_VEL
LIN {X 0,Y 368.85,Z 431.361,A -85,B 0,C 180,E1 -12781.092,E2 -12781.092} C_VEL
LIN {X 0,Y 368.937,Z 429.758,A -85,B 0,C 180,E1 -12782.183,E2 -12782.183} C_VEL
LIN {X 0,Y 368.806,Z 427.77,A -85,B 0,C 180,E1 -12783.277,E2 -12783.277} C_VEL
LIN {X 0,Y 369.264,Z 423.837,A -85,B 0,C 180,E1 -12784.913,E2 -12784.913} C_VEL
LIN {X 0,Y 369.493,Z 418.816,A -85,B 0,C 180,E1 -12786.553,E2 -12786.553} C_VEL
LIN {X 0,Y 370.071,Z 411.343,A -85,B 0,C 180,E1 -12788.463,E2 -12788.463} C_VEL
LIN {X 0,Y 370.545,Z 403.338,A -85,B 0,C 180,E1 -12790.104,E2 -12790.104} C_VEL
LIN {X 0,Y 371.215,Z 393.394,A -85,B 0,C 180,E1 -12791.743,E2 -12791.743} C_VEL
LIN {X 0,Y 371.87,Z 383.237,A -85,B 0,C 180,E1 -12793.108,E2 -12793.108} C_VEL
LIN {X 0,Y 372.565,Z 372.176,A -85,B 0,C 180,E1 -12794.31,E2 -12794.31} C_VEL
LIN {X 0,Y 372.852,Z 364.829,A -85,B 0,C 180,E1 -12794.992,E2 -12794.992} C_VEL
LIN {X 0,Y 369.687,Z 352.263,A -85,B 0,C 180,E1 -12796.071,E2 -12796.071} C_VEL
LIN {X 0,Y 369.019,Z 349.516,A -85,B 0,C 180,E1 -12796.314,E2 -12796.314} C_VEL
LIN {X 0,Y 368.938,Z 349.526,A -85,B 0,C 180,E1 -12800.053,E2 -12800.053} C_VEL
LIN {X 0,Y 368.948,Z 349.525,A -85,B 0,C 180,E1 -12803.887,E2 -12803.887} C_VEL
LIN {X 0,Y 368.971,Z 349.526,A -85,B 0,C 180,E1 -12807.203,E2 -12807.203} C_VEL
LIN {X 0,Y 368.921,Z 349.529,A -85,B 0,C 180,E1 -12809.69,E2 -12809.69} C_VEL
LIN {X 0,Y 368.899,Z 349.536,A -85,B 0,C 180,E1 -12813.043,E2 -12813.043} C_VEL
LIN {X 0,Y 368.92,Z 349.528,A -85,B 0,C 180,E1 -12816.196,E2 -12816.196} C_VEL
LIN {X 0,Y 368.911,Z 349.533,A -85,B 0,C 180,E1 -12818.952,E2 -12818.952} C_VEL
LIN {X 0,Y 368.911,Z 349.53,A -85,B 0,C 180,E1 -12822.014,E2 -12822.014} C_VEL
LIN {X 0,Y 368.909,Z 349.532,A -85,B 0,C 180,E1 -12825.18,E2 -12825.18} C_VEL
LIN {X 0,Y 368.885,Z 349.535,A -85,B 0,C 180,E1 -12828.178,E2 -12828.178} C_VEL
LIN {X 0,Y 368.91,Z 349.53,A -85,B 0,C 180,E1 -12831.359,E2 -12831.359} C_VEL
LIN {X 0,Y 368.937,Z 349.527,A -85,B 0,C 180,E1 -12835.146,E2 -12835.146} C_VEL
LIN {X 0,Y 368.93,Z 349.529,A -85,B 0,C 180,E1 -12839.046,E2 -12839.046} C_VEL
LIN {X 0,Y 368.964,Z 349.526,A -85,B 0,C 180,E1 -12842.796,E2 -12842.796} C_VEL
LIN {X 0,Y 368.946,Z 349.528,A -85,B 0,C 180,E1 -12846.113,E2 -12846.113} C_VEL
LIN {X 0,Y 368.946,Z 349.527,A -85,B 0,C 180,E1 -12849.947,E2 -12849.947} C_VEL
LIN {X 0,Y 368.977,Z 349.521,A -85,B 0,C 180,E1 -12853.399,E2 -12853.399} C_VEL
LIN {X 0,Y 369.058,Z 349.513,A -85,B 0,C 180,E1 -12856.79,E2 -12856.79} C_VEL
LIN {X 0,Y 369.068,Z 349.514,A -85,B 0,C 180,E1 -12860.132,E2 -12860.132} C_VEL
LIN {X 0,Y 369.2,Z 349.495,A -85,B 0,C 180,E1 -12863.442,E2 -12863.442} C_VEL
LIN {X 0,Y 369.32,Z 349.482,A -85,B 0,C 180,E1 -12867.819,E2 -12867.819} C_VEL
LIN {X 0,Y 369.458,Z 349.467,A -85,B 0,C 180,E1 -12870,E2 -12870} C_VEL
LIN {X 0,Y 369.32,Z 349.482,A -85,B 0,C 180,E1 -12872.181,E2 -12872.181} C_VEL
LIN {X 0,Y 369.2,Z 349.495,A -85,B 0,C 180,E1 -12876.558,E2 -12876.558} C_VEL
LIN {X 0,Y 369.069,Z 349.514,A -85,B 0,C 180,E1 -12879.868,E2 -12879.868} C_VEL
LIN {X 0,Y 369.038,Z 349.518,A -85,B 0,C 180,E1 -12883.773,E2 -12883.773} C_VEL
LIN {X 0,Y 369.002,Z 349.523,A -85,B 0,C 180,E1 -12887.769,E2 -12887.769} C_VEL
LIN {X 0,Y 368.931,Z 349.529,A -85,B 0,C 180,E1 -12891.22,E2 -12891.22} C_VEL
LIN {X 0,Y 368.959,Z 349.524,A -85,B 0,C 180,E1 -12894.776,E2 -12894.776} C_VEL
LIN {X 0,Y 368.964,Z 349.526,A -85,B 0,C 180,E1 -12897.204,E2 -12897.204} C_VEL
LIN {X 0,Y 368.93,Z 349.529,A -85,B 0,C 180,E1 -12900.954,E2 -12900.954} C_VEL
LIN {X 0,Y 368.93,Z 349.529,A -85,B 0,C 180,E1 -12905.002,E2 -12905.002} C_VEL
LIN {X 0,Y 368.911,Z 349.53,A -85,B 0,C 180,E1 -12908.641,E2 -12908.641} C_VEL
LIN {X 0,Y 368.943,Z 349.526,A -85,B 0,C 180,E1 -12912.02,E2 -12912.02} C_VEL
LIN {X 0,Y 368.93,Z 349.527,A -85,B 0,C 180,E1 -12912.232,E2 -12912.232} C_VEL
LIN {X 0,Y 368.227,Z 349.619,A -85,B 0,C 180,E1 -12913.142,E2 -12913.142} C_VEL
LIN {X 0,Y 365.326,Z 349.977,A -85,B 0,C 180,E1 -12914.622,E2 -12914.622} C_VEL
LIN {X 0,Y 362.906,Z 350.279,A -85,B 0,C 180,E1 -12915.82,E2 -12915.82} C_VEL
LIN {X 0,Y 361.899,Z 350.405,A -85,B 0,C 180,E1 -12916.747,E2 -12916.747} C_VEL
LIN {X 0,Y 361.833,Z 350.414,A -85,B 0,C 180,E1 -12917.06,E2 -12917.06} C_VEL
LIN {X 0,Y 361.872,Z 350.41,A -85,B 0,C 180,E1 -12920.974,E2 -12920.974} C_VEL
LIN {X 0,Y 361.877,Z 350.407,A -85,B 0,C 180,E1 -12924.656,E2 -12924.656} C_VEL
LIN {X 0,Y 361.84,Z 350.411,A -85,B 0,C 180,E1 -12928.371,E2 -12928.371} C_VEL
LIN {X 0,Y 361.903,Z 350.407,A -85,B 0,C 180,E1 -12930.956,E2 -12930.956} C_VEL
LIN {X 0,Y 361.958,Z 350.397,A -85,B 0,C 180,E1 -12933.476,E2 -12933.476} C_VEL
LIN {X 0,Y 361.894,Z 350.407,A -85,B 0,C 180,E1 -12937.145,E2 -12937.145} C_VEL
LIN {X 0,Y 361.911,Z 350.406,A -85,B 0,C 180,E1 -12940.724,E2 -12940.724} C_VEL
LIN {X 0,Y 361.937,Z 350.401,A -85,B 0,C 180,E1 -12943.066,E2 -12943.066} C_VEL
LIN {X 0,Y 362.003,Z 350.394,A -85,B 0,C 180,E1 -12946.528,E2 -12946.528} C_VEL
LIN {X 0,Y 362.036,Z 350.387,A -85,B 0,C 180,E1 -12949.938,E2 -12949.938} C_VEL
LIN {X 0,Y 362.156,Z 350.373,A -85,B 0,C 180,E1 -12952.193,E2 -12952.193} C_VEL
LIN {X 0,Y 362.122,Z 350.379,A -85,B 0,C 180,E1 -12954.431,E2 -12954.431} C_VEL
LIN {X 0,Y 362.285,Z 350.354,A -85,B 0,C 180,E1 -12957.777,E2 -12957.777} C_VEL
LIN {X 0,Y 362.431,Z 350.338,A -85,B 0,C 180,E1 -12960,E2 -12960} C_VEL
LIN {X 0,Y 362.288,Z 350.358,A -85,B 0,C 180,E1 -12962.224,E2 -12962.224} C_VEL
LIN {X 0,Y 362.153,Z 350.375,A -85,B 0,C 180,E1 -12966.687,E2 -12966.687} C_VEL
LIN {X 0,Y 362.033,Z 350.39,A -85,B 0,C 180,E1 -12970.062,E2 -12970.062} C_VEL
LIN {X 0,Y 362.002,Z 350.392,A -85,B 0,C 180,E1 -12973.899,E2 -12973.899} C_VEL
LIN {X 0,Y 361.972,Z 350.397,A -85,B 0,C 180,E1 -12977.939,E2 -12977.939} C_VEL
LIN {X 0,Y 361.897,Z 350.405,A -85,B 0,C 180,E1 -12981.653,E2 -12981.653} C_VEL
LIN {X 0,Y 361.933,Z 350.399,A -85,B 0,C 180,E1 -12985.29,E2 -12985.29} C_VEL
LIN {X 0,Y 361.923,Z 350.403,A -85,B 0,C 180,E1 -12987.778,E2 -12987.778} C_VEL
LIN {X 0,Y 361.851,Z 350.409,A -85,B 0,C 180,E1 -12991.285,E2 -12991.285} C_VEL
LIN {X 0,Y 361.859,Z 350.41,A -85,B 0,C 180,E1 -12994.28,E2 -12994.28} C_VEL
LIN {X 0,Y 361.869,Z 350.407,A -85,B 0,C 180,E1 -12997.223,E2 -12997.223} C_VEL
LIN {X 0,Y 361.839,Z 350.411,A -85,B 0,C 180,E1 -13000.755,E2 -13000.755} C_VEL
LIN {X 0,Y 361.898,Z 350.461,A -85,B 0,C 180,E1 -13004.649,E2 -13004.649} C_VEL
LIN {X 0,Y 363.839,Z 360.409,A -85,B 0,C 180,E1 -13008.461,E2 -13008.461} C_VEL
LIN {X 0,Y 365.739,Z 370.04,A -85,B 0,C 180,E1 -13011.986,E2 -13011.986} C_VEL
LIN {X 0,Y 365.905,Z 372.284,A -85,B 0,C 180,E1 -13012.769,E2 -13012.769} C_VEL
LIN {X 0,Y 364.576,Z 384.057,A -85,B 0,C 180,E1 -13016.674,E2 -13016.674} C_VEL
LIN {X 0,Y 363.518,Z 394.899,A -85,B 0,C 180,E1 -13020.209,E2 -13020.209} C_VEL
LIN {X 0,Y 362.501,Z 407.158,A -85,B 0,C 180,E1 -13024.137,E2 -13024.137} C_VEL
LIN {X 0,Y 361.752,Z 418.521,A -85,B 0,C 180,E1 -13027.738,E2 -13027.738} C_VEL
LIN {X 0,Y 361.317,Z 429.077,A -85,B 0,C 180,E1 -13031.059,E2 -13031.059} C_VEL
LIN {X 0,Y 362.364,Z 444.273,A -85,B 0,C 180,E1 -13031.715,E2 -13031.715} C_VEL
LIN {X 0,Y 363.261,Z 456.895,A -85,B 0,C 180,E1 -13032.477,E2 -13032.477} C_VEL
LIN {X 0,Y 363.905,Z 469.385,A -85,B 0,C 180,E1 -13033.449,E2 -13033.449} C_VEL
LIN {X 0,Y 363.9,Z 475.68,A -85,B 0,C 180,E1 -13034.025,E2 -13034.025} C_VEL
LIN {X 0,Y 362.928,Z 487.194,A -85,B 0,C 180,E1 -13035.276,E2 -13035.276} C_VEL
LIN {X 0,Y 362.204,Z 496.608,A -85,B 0,C 180,E1 -13036.535,E2 -13036.535} C_VEL
LIN {X 0,Y 361.665,Z 505.299,A -85,B 0,C 180,E1 -13037.942,E2 -13037.942} C_VEL
LIN {X 0,Y 361.243,Z 513.797,A -85,B 0,C 180,E1 -13039.632,E2 -13039.632} C_VEL
LIN {X 0,Y 361.108,Z 520.608,A -85,B 0,C 180,E1 -13041.325,E2 -13041.325} C_VEL
LIN {X 0,Y 361.137,Z 526.809,A -85,B 0,C 180,E1 -13043.294,E2 -13043.294} C_VEL
LIN {X 0,Y 361.383,Z 530.776,A -85,B 0,C 180,E1 -13044.979,E2 -13044.979} C_VEL
LIN {X 0,Y 361.434,Z 533.563,A -85,B 0,C 180,E1 -13046.656,E2 -13046.656} C_VEL
LIN {X 0,Y 361.488,Z 534.816,A -85,B 0,C 180,E1 -13047.771,E2 -13047.771} C_VEL
LIN {X 0,Y 361.68,Z 535.645,A -85,B 0,C 180,E1 -13048.886,E2 -13048.886} C_VEL
LIN {X 0,Y 361.851,Z 536.037,A -85,B 0,C 180,E1 -13050,E2 -13050} C_VEL
LIN {X 0,Y 361.694,Z 535.93,A -85,B 0,C 180,E1 -13051.113,E2 -13051.113} C_VEL
LIN {X 0,Y 361.353,Z 534.336,A -85,B 0,C 180,E1 -13053.345,E2 -13053.345} C_VEL
LIN {X 0,Y 361.292,Z 532.913,A -85,B 0,C 180,E1 -13054.463,E2 -13054.463} C_VEL
LIN {X 0,Y 361.068,Z 529.879,A -85,B 0,C 180,E1 -13056.146,E2 -13056.146} C_VEL
LIN {X 0,Y 360.928,Z 525.799,A -85,B 0,C 180,E1 -13057.834,E2 -13057.834} C_VEL
LIN {X 0,Y 361.013,Z 519.637,A -85,B 0,C 180,E1 -13059.808,E2 -13059.808} C_VEL
LIN {X 0,Y 361.488,Z 511.772,A -85,B 0,C 180,E1 -13061.779,E2 -13061.779} C_VEL
LIN {X 0,Y 362.197,Z 503.499,A -85,B 0,C 180,E1 -13063.465,E2 -13063.465} C_VEL
LIN {X 0,Y 363.11,Z 495.294,A -85,B 0,C 180,E1 -13064.86,E2 -13064.86} C_VEL
LIN {X 0,Y 364.452,Z 484.543,A -85,B 0,C 180,E1 -13066.381,E2 -13066.381} C_VEL
LIN {X 0,Y 365.555,Z 475.291,A -85,B 0,C 180,E1 -13067.482,E2 -13067.482} C_VEL
LIN {X 0,Y 366.101,Z 463.003,A -85,B 0,C 180,E1 -13068.757,E2 -13068.757} C_VEL
LIN {X 0,Y 366.422,Z 450.138,A -85,B 0,C 180,E1 -13069.874,E2 -13069.874} C_VEL
LIN {X 0,Y 365.53,Z 437.04,A -85,B 0,C 180,E1 -13070.889,E2 -13070.889} C_VEL
LIN {X 0,Y 363.347,Z 423.131,A -85,B 0,C 180,E1 -13071.895,E2 -13071.895} C_VEL
LIN {X 0,Y 361.584,Z 414.786,A -85,B 0,C 180,E1 -13072.482,E2 -13072.482} C_VEL
LIN {X 0,Y 362.221,Z 403.868,A -85,B 0,C 180,E1 -13075.885,E2 -13075.885} C_VEL
LIN {X 0,Y 363.214,Z 390.753,A -85,B 0,C 180,E1 -13080.205,E2 -13080.205} C_VEL
LIN {X 0,Y 364.421,Z 380.073,A -85,B 0,C 180,E1 -13084.006,E2 -13084.006} C_VEL
LIN {X 0,Y 365.86,Z 371.73,A -85,B 0,C 180,E1 -13087.236,E2 -13087.236} C_VEL
LIN {X 0,Y 365.584,Z 368.566,A -85,B 0,C 180,E1 -13088.666,E2 -13088.666} C_VEL
LIN {X 0,Y 364.413,Z 362.217,A -85,B 0,C 180,E1 -13091.963,E2 -13091.963} C_VEL
LIN {X 0,Y 363.316,Z 357.242,A -85,B 0,C 180,E1 -13095.085,E2 -13095.085} C_VEL
LIN {X 0,Y 362.34,Z 352.622,A -85,B 0,C 180,E1 -13098.74,E2 -13098.74} C_VEL
LIN {X 0,Y 361.873,Z 350.408,A -85,B 0,C 180,E1 -13100.973,E2 -13100.973} C_VEL
LIN {X 0,Y 361.878,Z 350.41,A -85,B 0,C 180,E1 -13104.655,E2 -13104.655} C_VEL
LIN {X 0,Y 361.841,Z 350.411,A -85,B 0,C 180,E1 -13108.371,E2 -13108.371} C_VEL
LIN {X 0,Y 361.903,Z 350.405,A -85,B 0,C 180,E1 -13110.955,E2 -13110.955} C_VEL
LIN {X 0,Y 361.958,Z 350.396,A -85,B 0,C 180,E1 -13113.475,E2 -13113.475} C_VEL
LIN {X 0,Y 361.894,Z 350.406,A -85,B 0,C 180,E1 -13117.145,E2 -13117.145} C_VEL
LIN {X 0,Y 362.933,Z 353.327,A -85,B 0,C 180,E1 -13117.479,E2 -13117.479} C_VEL
LIN {X 0,Y 363.795,Z 354.507,A -85,B 0,C 180,E1 -13117.669,E2 -13117.669} C_VEL
LIN {X 0,Y 369.087,Z 366.481,A -85,B 0,C 180,E1 -13119.286,E2 -13119.286} C_VEL
LIN {X 0,Y 371.792,Z 374.796,A -85,B 0,C 180,E1 -13120.425,E2 -13120.425} C_VEL
LIN {X 0,Y 372.263,Z 377.096,A -85,B 0,C 180,E1 -13120.728,E2 -13120.728} C_VEL
LIN {X 0,Y 370.967,Z 388.234,A -85,B 0,C 180,E1 -13121.985,E2 -13121.985} C_VEL
LIN {X 0,Y 369.75,Z 396.731,A -85,B 0,C 180,E1 -13123.15,E2 -13123.15} C_VEL
LIN {X 0,Y 368.532,Z 404.927,A -85,B 0,C 180,E1 -13124.515,E2 -13124.515} C_VEL
LIN {X 0,Y 367.138,Z 412.969,A -85,B 0,C 180,E1 -13126.156,E2 -13126.156} C_VEL
LIN {X 0,Y 365.964,Z 419.481,A -85,B 0,C 180,E1 -13127.804,E2 -13127.804} C_VEL
LIN {X 0,Y 364.976,Z 424.867,A -85,B 0,C 180,E1 -13129.542,E2 -13129.542} C_VEL
LIN {X 0,Y 364.063,Z 428.662,A -85,B 0,C 180,E1 -13131.116,E2 -13131.116} C_VEL
LIN {X 0,Y 363.6,Z 430.721,A -85,B 0,C 180,E1 -13132.224,E2 -13132.224} C_VEL
LIN {X 0,Y 363.136,Z 432.371,A -85,B 0,C 180,E1 -13133.331,E2 -13133.331} C_VEL
LIN {X 0,Y 362.826,Z 433.6,A -85,B 0,C 180,E1 -13134.442,E2 -13134.442} C_VEL
LIN {X 0,Y 362.575,Z 434.398,A -85,B 0,C 180,E1 -13135.553,E2 -13135.553} C_VEL
LIN {X 0,Y 362.176,Z 434.773,A -85,B 0,C 180,E1 -13137.776,E2 -13137.776} C_VEL
LIN {X 0,Y 362.047,Z 434.374,A -85,B 0,C 180,E1 -13138.888,E2 -13138.888} C_VEL
LIN {X 0,Y 361.977,Z 433.532,A -85,B 0,C 180,E1 -13140,E2 -13140} C_VEL
LIN {X 0,Y 361.825,Z 432.306,A -85,B 0,C 180,E1 -13141.113,E2 -13141.113} C_VEL
LIN {X 0,Y 361.821,Z 429.669,A -85,B 0,C 180,E1 -13142.783,E2 -13142.783} C_VEL
LIN {X 0,Y 361.953,Z 426.03,A -85,B 0,C 180,E1 -13144.454,E2 -13144.454} C_VEL
LIN {X 0,Y 362.238,Z 423.006,A -85,B 0,C 180,E1 -13145.567,E2 -13145.567} C_VEL
LIN {X 0,Y 362.686,Z 416.413,A -85,B 0,C 180,E1 -13147.516,E2 -13147.516} C_VEL
LIN {X 0,Y 363.229,Z 408.664,A -85,B 0,C 180,E1 -13149.323,E2 -13149.323} C_VEL
LIN {X 0,Y 363.761,Z 400.563,A -85,B 0,C 180,E1 -13150.858,E2 -13150.858} C_VEL
LIN {X 0,Y 364.455,Z 391.652,A -85,B 0,C 180,E1 -13152.246,E2 -13152.246} C_VEL
LIN {X 0,Y 365.132,Z 380.842,A -85,B 0,C 180,E1 -13153.638,E2 -13153.638} C_VEL
LIN {X 0,Y 365.761,Z 368.892,A -85,B 0,C 180,E1 -13154.877,E2 -13154.877} C_VEL
LIN {X 0,Y 365.832,Z 365.82,A -85,B 0,C 180,E1 -13155.159,E2 -13155.159} C_VEL
LIN {X 0,Y 362.754,Z 353.506,A -85,B 0,C 180,E1 -13156.243,E2 -13156.243} C_VEL
LIN {X 0,Y 361.973,Z 350.394,A -85,B 0,C 180,E1 -13156.496,E2 -13156.496} C_VEL
LIN {X 0,Y 361.896,Z 350.403,A -85,B 0,C 180,E1 -13160.46,E2 -13160.46} C_VEL
LIN {X 0,Y 361.898,Z 350.403,A -85,B 0,C 180,E1 -13164.114,E2 -13164.114} C_VEL
LIN {X 0,Y 361.945,Z 350.4,A -85,B 0,C 180,E1 -13166.722,E2 -13166.722} C_VEL
LIN {X 0,Y 361.877,Z 350.407,A -85,B 0,C 180,E1 -13170.328,E2 -13170.328} C_VEL
LIN {X 0,Y 361.856,Z 350.409,A -85,B 0,C 180,E1 -13174.28,E2 -13174.28} C_VEL
LIN {X 0,Y 361.868,Z 350.409,A -85,B 0,C 180,E1 -13177.223,E2 -13177.223} C_VEL
LIN {X 0,Y 361.875,Z 350.411,A -85,B 0,C 180,E1 -13180.762,E2 -13180.762} C_VEL
LIN {X 0,Y 361.841,Z 350.413,A -85,B 0,C 180,E1 -13184.365,E2 -13184.365} C_VEL
LIN {X 0,Y 361.838,Z 350.411,A -85,B 0,C 180,E1 -13187.568,E2 -13187.568} C_VEL
LIN {X 0,Y 361.871,Z 350.409,A -85,B 0,C 180,E1 -13190.973,E2 -13190.973} C_VEL
LIN {X 0,Y 361.875,Z 350.41,A -85,B 0,C 180,E1 -13194.655,E2 -13194.655} C_VEL
LIN {X 0,Y 361.838,Z 350.415,A -85,B 0,C 180,E1 -13198.37,E2 -13198.37} C_VEL
LIN {X 0,Y 361.909,Z 350.406,A -85,B 0,C 180,E1 -13202.221,E2 -13202.221} C_VEL
LIN {X 0,Y 361.929,Z 350.403,A -85,B 0,C 180,E1 -13204.71,E2 -13204.71} C_VEL
LIN {X 0,Y 361.9,Z 350.407,A -85,B 0,C 180,E1 -13208.347,E2 -13208.347} C_VEL
LIN {X 0,Y 361.968,Z 350.397,A -85,B 0,C 180,E1 -13212.061,E2 -13212.061} C_VEL
LIN {X 0,Y 361.998,Z 350.395,A -85,B 0,C 180,E1 -13216.101,E2 -13216.101} C_VEL
LIN {X 0,Y 362.032,Z 350.391,A -85,B 0,C 180,E1 -13219.938,E2 -13219.938} C_VEL
LIN {X 0,Y 362.162,Z 350.371,A -85,B 0,C 180,E1 -13223.314,E2 -13223.314} C_VEL
LIN {X 0,Y 362.284,Z 350.358,A -85,B 0,C 180,E1 -13227.777,E2 -13227.777} C_VEL
LIN {X 0,Y 362.427,Z 350.342,A -85,B 0,C 180,E1 -13230,E2 -13230} C_VEL
LIN {X 0,Y 362.284,Z 350.358,A -85,B 0,C 180,E1 -13232.224,E2 -13232.224} C_VEL
LIN {X 0,Y 362.162,Z 350.371,A -85,B 0,C 180,E1 -13236.686,E2 -13236.686} C_VEL
LIN {X 0,Y 362.033,Z 350.39,A -85,B 0,C 180,E1 -13240.062,E2 -13240.062} C_VEL
LIN {X 0,Y 361.999,Z 350.395,A -85,B 0,C 180,E1 -13243.899,E2 -13243.899} C_VEL
LIN {X 0,Y 361.968,Z 350.397,A -85,B 0,C 180,E1 -13247.939,E2 -13247.939} C_VEL
LIN {X 0,Y 361.894,Z 350.408,A -85,B 0,C 180,E1 -13251.653,E2 -13251.653} C_VEL
LIN {X 0,Y 361.93,Z 350.403,A -85,B 0,C 180,E1 -13255.29,E2 -13255.29} C_VEL
LIN {X 0,Y 361.909,Z 350.406,A -85,B 0,C 180,E1 -13257.779,E2 -13257.779} C_VEL
LIN {X 0,Y 361.839,Z 350.415,A -85,B 0,C 180,E1 -13261.63,E2 -13261.63} C_VEL
LIN {X 0,Y 361.876,Z 350.411,A -85,B 0,C 180,E1 -13265.345,E2 -13265.345} C_VEL
LIN {X 0,Y 361.874,Z 350.409,A -85,B 0,C 180,E1 -13269.027,E2 -13269.027} C_VEL
LIN {X 0,Y 361.885,Z 350.405,A -85,B 0,C 180,E1 -13272.441,E2 -13272.441} C_VEL
LIN {X 0,Y 361.849,Z 350.412,A -85,B 0,C 180,E1 -13275.637,E2 -13275.637} C_VEL
LIN {X 0,Y 361.833,Z 350.414,A -85,B 0,C 180,E1 -13277.06,E2 -13277.06} C_VEL
LIN {X 0,Y 361.198,Z 350.498,A -85,B 0,C 180,E1 -13277.989,E2 -13277.989} C_VEL
LIN {X 0,Y 358.323,Z 350.852,A -85,B 0,C 180,E1 -13279.498,E2 -13279.498} C_VEL
LIN {X 0,Y 355.884,Z 351.154,A -85,B 0,C 180,E1 -13280.72,E2 -13280.72} C_VEL
LIN {X 0,Y 354.866,Z 351.28,A -85,B 0,C 180,E1 -13281.665,E2 -13281.665} C_VEL
LIN {X 0,Y 354.8,Z 351.285,A -85,B 0,C 180,E1 -13281.986,E2 -13281.986} C_VEL
LIN {X 0,Y 354.815,Z 351.29,A -85,B 0,C 180,E1 -13284.941,E2 -13284.941} C_VEL
LIN {X 0,Y 354.796,Z 351.289,A -85,B 0,C 180,E1 -13288.405,E2 -13288.405} C_VEL
LIN {X 0,Y 354.854,Z 351.281,A -85,B 0,C 180,E1 -13291.619,E2 -13291.619} C_VEL
LIN {X 0,Y 354.903,Z 351.275,A -85,B 0,C 180,E1 -13294.173,E2 -13294.173} C_VEL
LIN {X 0,Y 354.838,Z 351.282,A -85,B 0,C 180,E1 -13297.894,E2 -13297.894} C_VEL
LIN {X 0,Y 354.926,Z 351.271,A -85,B 0,C 180,E1 -13301.892,E2 -13301.892} C_VEL
LIN {X 0,Y 354.947,Z 351.269,A -85,B 0,C 180,E1 -13305.981,E2 -13305.981} C_VEL
LIN {X 0,Y 354.983,Z 351.265,A -85,B 0,C 180,E1 -13309.736,E2 -13309.736} C_VEL
LIN {X 0,Y 355.119,Z 351.248,A -85,B 0,C 180,E1 -13312.037,E2 -13312.037} C_VEL
LIN {X 0,Y 355.097,Z 351.253,A -85,B 0,C 180,E1 -13314.321,E2 -13314.321} C_VEL
LIN {X 0,Y 355.248,Z 351.231,A -85,B 0,C 180,E1 -13317.733,E2 -13317.733} C_VEL
LIN {X 0,Y 355.401,Z 351.214,A -85,B 0,C 180,E1 -13320,E2 -13320} C_VEL
LIN {X 0,Y 355.251,Z 351.235,A -85,B 0,C 180,E1 -13322.268,E2 -13322.268} C_VEL
LIN {X 0,Y 355.116,Z 351.25,A -85,B 0,C 180,E1 -13326.82,E2 -13326.82} C_VEL
LIN {X 0,Y 354.981,Z 351.269,A -85,B 0,C 180,E1 -13330.264,E2 -13330.264} C_VEL
LIN {X 0,Y 354.948,Z 351.272,A -85,B 0,C 180,E1 -13334.019,E2 -13334.019} C_VEL
LIN {X 0,Y 354.927,Z 351.276,A -85,B 0,C 180,E1 -13338.109,E2 -13338.109} C_VEL
LIN {X 0,Y 354.839,Z 351.287,A -85,B 0,C 180,E1 -13342.106,E2 -13342.106} C_VEL
LIN {X 0,Y 354.904,Z 351.278,A -85,B 0,C 180,E1 -13345.827,E2 -13345.827} C_VEL
LIN {X 0,Y 354.858,Z 351.283,A -85,B 0,C 180,E1 -13349.678,E2 -13349.678} C_VEL
LIN {X 0,Y 354.81,Z 351.289,A -85,B 0,C 180,E1 -13353.702,E2 -13353.702} C_VEL
LIN {X 0,Y 354.803,Z 351.288,A -85,B 0,C 180,E1 -13356.459,E2 -13356.459} C_VEL
LIN {X 0,Y 354.827,Z 351.286,A -85,B 0,C 180,E1 -13359.424,E2 -13359.424} C_VEL
LIN {X 0,Y 354.793,Z 351.293,A -85,B 0,C 180,E1 -13362.867,E2 -13362.867} C_VEL
LIN {X 0,Y 354.862,Z 351.485,A -85,B 0,C 180,E1 -13364.421,E2 -13364.421} C_VEL
LIN {X 0,Y 356.892,Z 361.755,A -85,B 0,C 180,E1 -13368.444,E2 -13368.444} C_VEL
LIN {X 0,Y 358.566,Z 370.287,A -85,B 0,C 180,E1 -13371.63,E2 -13371.63} C_VEL
LIN {X 0,Y 358.912,Z 373.055,A -85,B 0,C 180,E1 -13372.625,E2 -13372.625} C_VEL
LIN {X 0,Y 357.544,Z 384.802,A -85,B 0,C 180,E1 -13376.607,E2 -13376.607} C_VEL
LIN {X 0,Y 356.34,Z 396.377,A -85,B 0,C 180,E1 -13380.457,E2 -13380.457} C_VEL
LIN {X 0,Y 355.398,Z 407.816,A -85,B 0,C 180,E1 -13384.211,E2 -13384.211} C_VEL
LIN {X 0,Y 354.633,Z 419.105,A -85,B 0,C 180,E1 -13387.88,E2 -13387.88} C_VEL
LIN {X 0,Y 354.23,Z 428.214,A -85,B 0,C 180,E1 -13390.816,E2 -13390.816} C_VEL
LIN {X 0,Y 355.226,Z 443.048,A -85,B 0,C 180,E1 -13391.47,E2 -13391.47} C_VEL
LIN {X 0,Y 356.098,Z 455.739,A -85,B 0,C 180,E1 -13392.248,E2 -13392.248} C_VEL
LIN {X 0,Y 356.771,Z 468.415,A -85,B 0,C 180,E1 -13393.256,E2 -13393.256} C_VEL
LIN {X 0,Y 356.904,Z 474.747,A -85,B 0,C 180,E1 -13393.85,E2 -13393.85} C_VEL
LIN {X 0,Y 355.918,Z 486.228,A -85,B 0,C 180,E1 -13395.125,E2 -13395.125} C_VEL
LIN {X 0,Y 355.118,Z 496.579,A -85,B 0,C 180,E1 -13396.553,E2 -13396.553} C_VEL
LIN {X 0,Y 354.572,Z 505.097,A -85,B 0,C 180,E1 -13397.988,E2 -13397.988} C_VEL
LIN {X 0,Y 354.178,Z 513.402,A -85,B 0,C 180,E1 -13399.712,E2 -13399.712} C_VEL
LIN {X 0,Y 354.07,Z 520.092,A -85,B 0,C 180,E1 -13401.438,E2 -13401.438} C_VEL
LIN {X 0,Y 354.099,Z 525.381,A -85,B 0,C 180,E1 -13403.161,E2 -13403.161} C_VEL
LIN {X 0,Y 354.349,Z 529.442,A -85,B 0,C 180,E1 -13404.879,E2 -13404.879} C_VEL
LIN {X 0,Y 354.415,Z 532.308,A -85,B 0,C 180,E1 -13406.589,E2 -13406.589} C_VEL
LIN {X 0,Y 354.469,Z 533.63,A -85,B 0,C 180,E1 -13407.727,E2 -13407.727} C_VEL
LIN {X 0,Y 354.681,Z 534.491,A -85,B 0,C 180,E1 -13408.865,E2 -13408.865} C_VEL
LIN {X 0,Y 354.839,Z 534.911,A -85,B 0,C 180,E1 -13410,E2 -13410} C_VEL
LIN {X 0,Y 354.664,Z 534.846,A -85,B 0,C 180,E1 -13411.135,E2 -13411.135} C_VEL
LIN {X 0,Y 354.377,Z 534.296,A -85,B 0,C 180,E1 -13412.273,E2 -13412.273} C_VEL
LIN {X 0,Y 354.301,Z 533.325,A -85,B 0,C 180,E1 -13413.412,E2 -13413.412} C_VEL
LIN {X 0,Y 354.218,Z 531.93,A -85,B 0,C 180,E1 -13414.552,E2 -13414.552} C_VEL
LIN {X 0,Y 353.947,Z 528.477,A -85,B 0,C 180,E1 -13416.511,E2 -13416.511} C_VEL
LIN {X 0,Y 353.839,Z 523.388,A -85,B 0,C 180,E1 -13418.567,E2 -13418.567} C_VEL
LIN {X 0,Y 354.039,Z 516.853,A -85,B 0,C 180,E1 -13420.581,E2 -13420.581} C_VEL
LIN {X 0,Y 354.595,Z 509.933,A -85,B 0,C 180,E1 -13422.302,E2 -13422.302} C_VEL
LIN {X 0,Y 355.363,Z 501.067,A -85,B 0,C 180,E1 -13424.113,E2 -13424.113} C_VEL
LIN {X 0,Y 356.674,Z 491.419,A -85,B 0,C 180,E1 -13425.72,E2 -13425.72} C_VEL
LIN {X 0,Y 358.283,Z 480.247,A -85,B 0,C 180,E1 -13427.259,E2 -13427.259} C_VEL
LIN {X 0,Y 359.041,Z 470.593,A -85,B 0,C 180,E1 -13428.399,E2 -13428.399} C_VEL
LIN {X 0,Y 359.784,Z 458.036,A -85,B 0,C 180,E1 -13429.66,E2 -13429.66} C_VEL
LIN {X 0,Y 359.686,Z 445.277,A -85,B 0,C 180,E1 -13430.781,E2 -13430.781} C_VEL
LIN {X 0,Y 358.329,Z 431.716,A -85,B 0,C 180,E1 -13431.879,E2 -13431.879} C_VEL
LIN {X 0,Y 355.568,Z 417.372,A -85,B 0,C 180,E1 -13432.982,E2 -13432.982} C_VEL
LIN {X 0,Y 354.641,Z 412.858,A -85,B 0,C 180,E1 -13433.35,E2 -13433.35} C_VEL
LIN {X 0,Y 355.272,Z 403.296,A -85,B 0,C 180,E1 -13436.43,E2 -13436.43} C_VEL
LIN {X 0,Y 356.221,Z 392.151,A -85,B 0,C 180,E1 -13440.21,E2 -13440.21} C_VEL
LIN {X 0,Y 357.589,Z 380.803,A -85,B 0,C 180,E1 -13444.364,E2 -13444.364} C_VEL
LIN {X 0,Y 358.972,Z 373.276,A -85,B 0,C 180,E1 -13447.368,E2 -13447.368} C_VEL
LIN {X 0,Y 358.489,Z 368.875,A -85,B 0,C 180,E1 -13449.451,E2 -13449.451} C_VEL
LIN {X 0,Y 357.401,Z 363.157,A -85,B 0,C 180,E1 -13452.604,E2 -13452.604} C_VEL
LIN {X 0,Y 356.167,Z 357.682,A -85,B 0,C 180,E1 -13456.32,E2 -13456.32} C_VEL
LIN {X 0,Y 355.472,Z 354.205,A -85,B 0,C 180,E1 -13459.274,E2 -13459.274} C_VEL
LIN {X 0,Y 354.817,Z 351.288,A -85,B 0,C 180,E1 -13462.682,E2 -13462.682} C_VEL
LIN {X 0,Y 354.834,Z 351.287,A -85,B 0,C 180,E1 -13466.318,E2 -13466.318} C_VEL
LIN {X 0,Y 354.872,Z 351.279,A -85,B 0,C 180,E1 -13470.621,E2 -13470.621} C_VEL
LIN {X 0,Y 354.903,Z 351.278,A -85,B 0,C 180,E1 -13474.173,E2 -13474.173} C_VEL
LIN {X 0,Y 354.875,Z 351.415,A -85,B 0,C 180,E1 -13476.275,E2 -13476.275} C_VEL
LIN {X 0,Y 355.924,Z 354.256,A -85,B 0,C 180,E1 -13476.622,E2 -13476.622} C_VEL
LIN {X 0,Y 358.187,Z 358.387,A -85,B 0,C 180,E1 -13477.249,E2 -13477.249} C_VEL
LIN {X 0,Y 362.361,Z 367.533,A -85,B 0,C 180,E1 -13478.586,E2 -13478.586} C_VEL
LIN {X 0,Y 365.704,Z 377.436,A -85,B 0,C 180,E1 -13480.022,E2 -13480.022} C_VEL
LIN {X 0,Y 365.977,Z 380.204,A -85,B 0,C 180,E1 -13480.383,E2 -13480.383} C_VEL
LIN {X 0,Y 364.727,Z 389.815,A -85,B 0,C 180,E1 -13481.522,E2 -13481.522} C_VEL
LIN {X 0,Y 363.29,Z 399.087,A -85,B 0,C 180,E1 -13482.841,E2 -13482.841} C_VEL
LIN {X 0,Y 361.73,Z 408.497,A -85,B 0,C 180,E1 -13484.505,E2 -13484.505} C_VEL
LIN {X 0,Y 360.299,Z 416.095,A -85,B 0,C 180,E1 -13486.175,E2 -13486.175} C_VEL
LIN {X 0,Y 359.014,Z 422.524,A -85,B 0,C 180,E1 -13487.98,E2 -13487.98} C_VEL
LIN {X 0,Y 357.847,Z 427.683,A -85,B 0,C 180,E1 -13489.819,E2 -13489.819} C_VEL
LIN {X 0,Y 357.214,Z 430.187,A -85,B 0,C 180,E1 -13490.944,E2 -13490.944} C_VEL
LIN {X 0,Y 356.738,Z 432.169,A -85,B 0,C 180,E1 -13492.073,E2 -13492.073} C_VEL
LIN {X 0,Y 356.227,Z 433.757,A -85,B 0,C 180,E1 -13493.202,E2 -13493.202} C_VEL
LIN {X 0,Y 355.897,Z 434.91,A -85,B 0,C 180,E1 -13494.333,E2 -13494.333} C_VEL
LIN {X 0,Y 355.355,Z 435.952,A -85,B 0,C 180,E1 -13496.598,E2 -13496.598} C_VEL
LIN {X 0,Y 355.17,Z 435.897,A -85,B 0,C 180,E1 -13497.732,E2 -13497.732} C_VEL
LIN {X 0,Y 355.029,Z 435.426,A -85,B 0,C 180,E1 -13498.866,E2 -13498.866} C_VEL
LIN {X 0,Y 354.955,Z 434.525,A -85,B 0,C 180,E1 -13500,E2 -13500} C_VEL
LIN {X 0,Y 354.799,Z 433.243,A -85,B 0,C 180,E1 -13501.135,E2 -13501.135} C_VEL
LIN {X 0,Y 354.788,Z 430.508,A -85,B 0,C 180,E1 -13502.838,E2 -13502.838} C_VEL
LIN {X 0,Y 354.924,Z 426.767,A -85,B 0,C 180,E1 -13504.543,E2 -13504.543} C_VEL
LIN {X 0,Y 355.388,Z 421.914,A -85,B 0,C 180,E1 -13506.244,E2 -13506.244} C_VEL
LIN {X 0,Y 355.728,Z 415.873,A -85,B 0,C 180,E1 -13507.949,E2 -13507.949} C_VEL
LIN {X 0,Y 356.31,Z 408.384,A -85,B 0,C 180,E1 -13509.651,E2 -13509.651} C_VEL
LIN {X 0,Y 356.885,Z 399.149,A -85,B 0,C 180,E1 -13511.357,E2 -13511.357} C_VEL
LIN {X 0,Y 357.675,Z 389.774,A -85,B 0,C 180,E1 -13512.771,E2 -13512.771} C_VEL
LIN {X 0,Y 358.306,Z 379.5,A -85,B 0,C 180,E1 -13514.048,E2 -13514.048} C_VEL
LIN {X 0,Y 358.818,Z 368.049,A -85,B 0,C 180,E1 -13515.216,E2 -13515.216} C_VEL
LIN {X 0,Y 358.429,Z 365.303,A -85,B 0,C 180,E1 -13515.48,E2 -13515.48} C_VEL
LIN {X 0,Y 355.233,Z 352.617,A -85,B 0,C 180,E1 -13516.597,E2 -13516.597} C_VEL
LIN {X 0,Y 354.916,Z 351.274,A -85,B 0,C 180,E1 -13516.723,E2 -13516.723} C_VEL
LIN {X 0,Y 354.86,Z 351.281,A -85,B 0,C 180,E1 -13519.675,E2 -13519.675} C_VEL
LIN {X 0,Y 354.835,Z 351.286,A -85,B 0,C 180,E1 -13523.336,E2 -13523.336} C_VEL
LIN {X 0,Y 354.891,Z 351.28,A -85,B 0,C 180,E1 -13526.982,E2 -13526.982} C_VEL
LIN {X 0,Y 354.856,Z 351.281,A -85,B 0,C 180,E1 -13529.678,E2 -13529.678} C_VEL
LIN {X 0,Y 354.808,Z 351.286,A -85,B 0,C 180,E1 -13533.702,E2 -13533.702} C_VEL
LIN {X 0,Y 354.801,Z 351.288,A -85,B 0,C 180,E1 -13536.459,E2 -13536.459} C_VEL
LIN {X 0,Y 354.826,Z 351.285,A -85,B 0,C 180,E1 -13539.423,E2 -13539.423} C_VEL
LIN {X 0,Y 354.806,Z 351.291,A -85,B 0,C 180,E1 -13542.87,E2 -13542.87} C_VEL
LIN {X 0,Y 354.777,Z 351.291,A -85,B 0,C 180,E1 -13546.105,E2 -13546.105} C_VEL
LIN {X 0,Y 354.79,Z 351.29,A -85,B 0,C 180,E1 -13549.179,E2 -13549.179} C_VEL
LIN {X 0,Y 354.812,Z 351.289,A -85,B 0,C 180,E1 -13552.401,E2 -13552.401} C_VEL
LIN {X 0,Y 354.813,Z 351.288,A -85,B 0,C 180,E1 -13554.941,E2 -13554.941} C_VEL
LIN {X 0,Y 354.794,Z 351.293,A -85,B 0,C 180,E1 -13558.405,E2 -13558.405} C_VEL
LIN {X 0,Y 354.847,Z 351.282,A -85,B 0,C 180,E1 -13561.619,E2 -13561.619} C_VEL
